LIN {X 0,Y 249.082,Z 599.459,A -85,B 0,C 180,E1 -18921.519,E2 -18921.519} C_VEL
LIN {X 0,Y 249.126,Z 599.438,A -85,B 0,C 180,E1 -18925.483,E2 -18925.483} C_VEL
LIN {X 0,Y 249.079,Z 599.446,A -85,B 0,C 180,E1 -18928.994,E2 -18928.994} C_VEL
LIN {X 0,Y 249.033,Z 599.465,A -85,B 0,C 180,E1 -18932.426,E2 -18932.426} C_VEL
LIN {X 0,Y 249.071,Z 599.46,A -85,B 0,C 180,E1 -18936.339,E2 -18936.339} C_VEL
LIN {X 0,Y 249.033,Z 599.471,A -85,B 0,C 180,E1 -18940.94,E2 -18940.94} C_VEL
LIN {X 0,Y 249.934,Z 602.079,A -85,B 0,C 180,E1 -18941.228,E2 -18941.228} C_VEL
LIN {X 0,Y 251.998,Z 604.708,A -85,B 0,C 180,E1 -18941.748,E2 -18941.748} C_VEL
LIN {X 0,Y 262.179,Z 620.888,A -85,B 0,C 180,E1 -18944.251,E2 -18944.251} C_VEL
LIN {X 0,Y 269.73,Z 634.216,A -85,B 0,C 180,E1 -18945.97,E2 -18945.97} C_VEL
LIN {X 0,Y 273.492,Z 641.681,A -85,B 0,C 180,E1 -18946.804,E2 -18946.804} C_VEL
LIN {X 0,Y 271.471,Z 691.803,A -85,B 0,C 180,E1 -18948.109,E2 -18948.109} C_VEL
LIN {X 0,Y 270.735,Z 705.187,A -85,B 0,C 180,E1 -18948.696,E2 -18948.696} C_VEL
LIN {X 0,Y 269.486,Z 718.044,A -85,B 0,C 180,E1 -18949.556,E2 -18949.556} C_VEL
LIN {X 0,Y 267.657,Z 730.406,A -85,B 0,C 180,E1 -18950.695,E2 -18950.695} C_VEL
LIN {X 0,Y 265.617,Z 741.459,A -85,B 0,C 180,E1 -18952.037,E2 -18952.037} C_VEL
LIN {X 0,Y 263.18,Z 752.351,A -85,B 0,C 180,E1 -18953.717,E2 -18953.717} C_VEL
LIN {X 0,Y 260.708,Z 761.621,A -85,B 0,C 180,E1 -18955.522,E2 -18955.522} C_VEL
LIN {X 0,Y 258.17,Z 770.535,A -85,B 0,C 180,E1 -18957.713,E2 -18957.713} C_VEL
LIN {X 0,Y 255.828,Z 777.697,A -85,B 0,C 180,E1 -18959.911,E2 -18959.911} C_VEL
LIN {X 0,Y 253.498,Z 784.302,A -85,B 0,C 180,E1 -18962.52,E2 -18962.52} C_VEL
LIN {X 0,Y 251.573,Z 789.492,A -85,B 0,C 180,E1 -18965.226,E2 -18965.226} C_VEL
LIN {X 0,Y 250.056,Z 793.37,A -85,B 0,C 180,E1 -18968.047,E2 -18968.047} C_VEL
LIN {X 0,Y 249.088,Z 795.421,A -85,B 0,C 180,E1 -18970.21,E2 -18970.21} C_VEL
LIN {X 0,Y 248.544,Z 796.494,A -85,B 0,C 180,E1 -18971.878,E2 -18971.878} C_VEL
LIN {X 0,Y 247.872,Z 797.374,A -85,B 0,C 180,E1 -18975.216,E2 -18975.216} C_VEL
LIN {X 0,Y 247.669,Z 797.218,A -85,B 0,C 180,E1 -18976.879,E2 -18976.879} C_VEL
LIN {X 0,Y 247.624,Z 795.63,A -85,B 0,C 180,E1 -18980.196,E2 -18980.196} C_VEL
LIN {X 0,Y 247.906,Z 793.165,A -85,B 0,C 180,E1 -18982.855,E2 -18982.855} C_VEL
LIN {X 0,Y 248.296,Z 790.13,A -85,B 0,C 180,E1 -18985.129,E2 -18985.129} C_VEL
LIN {X 0,Y 248.985,Z 785.826,A -85,B 0,C 180,E1 -18987.573,E2 -18987.573} C_VEL
LIN {X 0,Y 249.851,Z 780.356,A -85,B 0,C 180,E1 -18990,E2 -18990} C_VEL
LIN {X 0,Y 251.008,Z 773.505,A -85,B 0,C 180,E1 -18992.407,E2 -18992.407} C_VEL
LIN {X 0,Y 252.54,Z 764.911,A -85,B 0,C 180,E1 -18994.789,E2 -18994.789} C_VEL
LIN {X 0,Y 254.059,Z 756.117,A -85,B 0,C 180,E1 -18996.752,E2 -18996.752} C_VEL
LIN {X 0,Y 255.471,Z 746.489,A -85,B 0,C 180,E1 -18998.503,E2 -18998.503} C_VEL
LIN {X 0,Y 257.112,Z 734.896,A -85,B 0,C 180,E1 -19000.154,E2 -19000.154} C_VEL
LIN {X 0,Y 258.501,Z 722.796,A -85,B 0,C 180,E1 -19001.49,E2 -19001.49} C_VEL
LIN {X 0,Y 259.536,Z 710.236,A -85,B 0,C 180,E1 -19002.511,E2 -19002.511} C_VEL
LIN {X 0,Y 260.222,Z 696.894,A -85,B 0,C 180,E1 -19003.262,E2 -19003.262} C_VEL
LIN {X 0,Y 260.83,Z 676.4,A -85,B 0,C 180,E1 -19003.888,E2 -19003.888} C_VEL
LIN {X 0,Y 262.109,Z 629.666,A -85,B 0,C 180,E1 -19005.142,E2 -19005.142} C_VEL
LIN {X 0,Y 253.908,Z 610.003,A -85,B 0,C 180,E1 -19006.539,E2 -19006.539} C_VEL
LIN {X 0,Y 252.057,Z 606.531,A -85,B 0,C 180,E1 -19006.849,E2 -19006.849} C_VEL
LIN {X 0,Y 261.743,Z 629.406,A -85,B 0,C 180,E1 -19008.542,E2 -19008.542} C_VEL
LIN {X 0,Y 262.782,Z 631.947,A -85,B 0,C 180,E1 -19008.719,E2 -19008.719} C_VEL
LIN {X 0,Y 260.482,Z 693.854,A -85,B 0,C 180,E1 -19010.636,E2 -19010.636} C_VEL
LIN {X 0,Y 259.825,Z 707.287,A -85,B 0,C 180,E1 -19011.365,E2 -19011.365} C_VEL
LIN {X 0,Y 258.74,Z 719.997,A -85,B 0,C 180,E1 -19012.35,E2 -19012.35} C_VEL
LIN {X 0,Y 257.533,Z 731.237,A -85,B 0,C 180,E1 -19013.522,E2 -19013.522} C_VEL
LIN {X 0,Y 255.956,Z 743.817,A -85,B 0,C 180,E1 -19015.219,E2 -19015.219} C_VEL
LIN {X 0,Y 254.453,Z 753.674,A -85,B 0,C 180,E1 -19016.889,E2 -19016.889} C_VEL
LIN {X 0,Y 252.923,Z 763.074,A -85,B 0,C 180,E1 -19018.868,E2 -19018.868} C_VEL
LIN {X 0,Y 251.449,Z 771.778,A -85,B 0,C 180,E1 -19021.134,E2 -19021.134} C_VEL
LIN {X 0,Y 250.227,Z 778.82,A -85,B 0,C 180,E1 -19023.406,E2 -19023.406} C_VEL
LIN {X 0,Y 249.306,Z 784.585,A -85,B 0,C 180,E1 -19025.718,E2 -19025.718} C_VEL
LIN {X 0,Y 248.469,Z 789.922,A -85,B 0,C 180,E1 -19028.481,E2 -19028.481} C_VEL
LIN {X 0,Y 247.942,Z 793.177,A -85,B 0,C 180,E1 -19030.687,E2 -19030.687} C_VEL
LIN {X 0,Y 247.595,Z 795.616,A -85,B 0,C 180,E1 -19032.939,E2 -19032.939} C_VEL
LIN {X 0,Y 247.507,Z 797.247,A -85,B 0,C 180,E1 -19035.224,E2 -19035.224} C_VEL
LIN {X 0,Y 247.614,Z 798.097,A -85,B 0,C 180,E1 -19037.556,E2 -19037.556} C_VEL
LIN {X 0,Y 247.975,Z 798.121,A -85,B 0,C 180,E1 -19039.925,E2 -19039.925} C_VEL
LIN {X 0,Y 248.631,Z 797.271,A -85,B 0,C 180,E1 -19042.321,E2 -19042.321} C_VEL
LIN {X 0,Y 249.53,Z 795.476,A -85,B 0,C 180,E1 -19044.762,E2 -19044.762} C_VEL
LIN {X 0,Y 251.057,Z 791.727,A -85,B 0,C 180,E1 -19047.867,E2 -19047.867} C_VEL
LIN {X 0,Y 252.676,Z 787.333,A -85,B 0,C 180,E1 -19050.416,E2 -19050.416} C_VEL
LIN {X 0,Y 254.848,Z 781.199,A -85,B 0,C 180,E1 -19053.079,E2 -19053.079} C_VEL
LIN {X 0,Y 257.014,Z 774.612,A -85,B 0,C 180,E1 -19055.293,E2 -19055.293} C_VEL
LIN {X 0,Y 259.391,Z 766.758,A -85,B 0,C 180,E1 -19057.406,E2 -19057.406} C_VEL
LIN {X 0,Y 261.928,Z 757.594,A -85,B 0,C 180,E1 -19059.38,E2 -19059.38} C_VEL
LIN {X 0,Y 264.28,Z 747.756,A -85,B 0,C 180,E1 -19061.087,E2 -19061.087} C_VEL
LIN {X 0,Y 264.764,Z 743.074,A -85,B 0,C 180,E1 -19061.862,E2 -19061.862} C_VEL
LIN {X 0,Y 263.45,Z 732.357,A -85,B 0,C 180,E1 -19063.76,E2 -19063.76} C_VEL
LIN {X 0,Y 262.988,Z 725.778,A -85,B 0,C 180,E1 -19064.699,E2 -19064.699} C_VEL
LIN {X 0,Y 263.253,Z 722.241,A -85,B 0,C 180,E1 -19065.063,E2 -19065.063} C_VEL
LIN {X 0,Y 264.76,Z 709.401,A -85,B 0,C 180,E1 -19066.034,E2 -19066.034} C_VEL
LIN {X 0,Y 265.703,Z 696.323,A -85,B 0,C 180,E1 -19066.707,E2 -19066.707} C_VEL
LIN {X 0,Y 268.808,Z 643.586,A -85,B 0,C 180,E1 -19068.39,E2 -19068.39} C_VEL
LIN {X 0,Y 262.795,Z 631.883,A -85,B 0,C 180,E1 -19070.124,E2 -19070.124} C_VEL
LIN {X 0,Y 255.885,Z 620.412,A -85,B 0,C 180,E1 -19072.262,E2 -19072.262} C_VEL
LIN {X 0,Y 251.655,Z 613.959,A -85,B 0,C 180,E1 -19073.687,E2 -19073.687} C_VEL
LIN {X 0,Y 248.959,Z 610.142,A -85,B 0,C 180,E1 -19074.634,E2 -19074.634} C_VEL
LIN {X 0,Y 246.533,Z 607.111,A -85,B 0,C 180,E1 -19075.512,E2 -19075.512} C_VEL
LIN {X 0,Y 245.545,Z 605.398,A -85,B 0,C 180,E1 -19075.914,E2 -19075.914} C_VEL
LIN {X 0,Y 243.492,Z 603.287,A -85,B 0,C 180,E1 -19076.691,E2 -19076.691} C_VEL
LIN {X 0,Y 242.539,Z 600.953,A -85,B 0,C 180,E1 -19077.145,E2 -19077.145} C_VEL
LIN {X 0,Y 242.441,Z 600.281,A -85,B 0,C 180,E1 -19077.3,E2 -19077.3} C_VEL
LIN {X 0,Y 242.692,Z 600.249,A -85,B 0,C 180,E1 -19080,E2 -19080} C_VEL
LIN {X 0,Y 242.631,Z 600.261,A -85,B 0,C 180,E1 -19081.66,E2 -19081.66} C_VEL
LIN {X 0,Y 242.427,Z 600.277,A -85,B 0,C 180,E1 -19086.659,E2 -19086.659} C_VEL
LIN {X 0,Y 242.309,Z 600.288,A -85,B 0,C 180,E1 -19090.022,E2 -19090.022} C_VEL
LIN {X 0,Y 242.151,Z 600.315,A -85,B 0,C 180,E1 -19095.142,E2 -19095.142} C_VEL
LIN {X 0,Y 242.066,Z 600.326,A -85,B 0,C 180,E1 -19098.625,E2 -19098.625} C_VEL
LIN {X 0,Y 242.008,Z 600.337,A -85,B 0,C 180,E1 -19102.18,E2 -19102.18} C_VEL
LIN {X 0,Y 242.063,Z 600.334,A -85,B 0,C 180,E1 -19105.839,E2 -19105.839} C_VEL
LIN {X 0,Y 242.026,Z 600.335,A -85,B 0,C 180,E1 -19109.581,E2 -19109.581} C_VEL
LIN {X 0,Y 241.988,Z 600.335,A -85,B 0,C 180,E1 -19113.492,E2 -19113.492} C_VEL
LIN {X 0,Y 242.01,Z 600.338,A -85,B 0,C 180,E1 -19117.578,E2 -19117.578} C_VEL
LIN {X 0,Y 242.016,Z 600.535,A -85,B 0,C 180,E1 -19118.962,E2 -19118.962} C_VEL
LIN {X 0,Y 243.784,Z 605.815,A -85,B 0,C 180,E1 -19122.647,E2 -19122.647} C_VEL
LIN {X 0,Y 245.968,Z 612.642,A -85,B 0,C 180,E1 -19126.707,E2 -19126.707} C_VEL
LIN {X 0,Y 247.835,Z 619.474,A -85,B 0,C 180,E1 -19130.189,E2 -19130.189} C_VEL
LIN {X 0,Y 250.568,Z 624.665,A -85,B 0,C 180,E1 -19131.241,E2 -19131.241} C_VEL
LIN {X 0,Y 252.18,Z 627.583,A -85,B 0,C 180,E1 -19131.822,E2 -19131.822} C_VEL
LIN {X 0,Y 255.009,Z 632.985,A -85,B 0,C 180,E1 -19132.801,E2 -19132.801} C_VEL
LIN {X 0,Y 259.392,Z 642.122,A -85,B 0,C 180,E1 -19134.256,E2 -19134.256} C_VEL
LIN {X 0,Y 262.407,Z 649.312,A -85,B 0,C 180,E1 -19135.233,E2 -19135.233} C_VEL
LIN {X 0,Y 264.894,Z 668.043,A -85,B 0,C 180,E1 -19136.557,E2 -19136.557} C_VEL
LIN {X 0,Y 266.173,Z 683.879,A -85,B 0,C 180,E1 -19137.483,E2 -19137.483} C_VEL
LIN {X 0,Y 266.569,Z 690.964,A -85,B 0,C 180,E1 -19137.858,E2 -19137.858} C_VEL
LIN {X 0,Y 263.985,Z 733.939,A -85,B 0,C 180,E1 -19139.233,E2 -19139.233} C_VEL
LIN {X 0,Y 262.386,Z 747.924,A -85,B 0,C 180,E1 -19139.965,E2 -19139.965} C_VEL
LIN {X 0,Y 260.203,Z 760.61,A -85,B 0,C 180,E1 -19140.911,E2 -19140.911} C_VEL
LIN {X 0,Y 257.602,Z 772.84,A -85,B 0,C 180,E1 -19142.147,E2 -19142.147} C_VEL
LIN {X 0,Y 254.816,Z 783.944,A -85,B 0,C 180,E1 -19143.594,E2 -19143.594} C_VEL
LIN {X 0,Y 252.114,Z 794.049,A -85,B 0,C 180,E1 -19145.283,E2 -19145.283} C_VEL
LIN {X 0,Y 249.332,Z 803.305,A -85,B 0,C 180,E1 -19147.197,E2 -19147.197} C_VEL
LIN {X 0,Y 246.566,Z 812.457,A -85,B 0,C 180,E1 -19149.564,E2 -19149.564} C_VEL
LIN {X 0,Y 244.524,Z 819.897,A -85,B 0,C 180,E1 -19152.003,E2 -19152.003} C_VEL
LIN {X 0,Y 242.872,Z 824.973,A -85,B 0,C 180,E1 -19154.044,E2 -19154.044} C_VEL
LIN {X 0,Y 241.494,Z 829.974,A -85,B 0,C 180,E1 -19156.537,E2 -19156.537} C_VEL
LIN {X 0,Y 240.654,Z 833.88,A -85,B 0,C 180,E1 -19159.058,E2 -19159.058} C_VEL
LIN {X 0,Y 240.244,Z 836.788,A -85,B 0,C 180,E1 -19161.589,E2 -19161.589} C_VEL
LIN {X 0,Y 240.238,Z 838.715,A -85,B 0,C 180,E1 -19164.07,E2 -19164.07} C_VEL
LIN {X 0,Y 240.322,Z 839.767,A -85,B 0,C 180,E1 -19166.647,E2 -19166.647} C_VEL
LIN {X 0,Y 240.609,Z 839.94,A -85,B 0,C 180,E1 -19168.326,E2 -19168.326} C_VEL
LIN {X 0,Y 240.759,Z 839.692,A -85,B 0,C 180,E1 -19170,E2 -19170} C_VEL
LIN {X 0,Y 240.697,Z 838.969,A -85,B 0,C 180,E1 -19171.673,E2 -19171.673} C_VEL
LIN {X 0,Y 240.236,Z 837.756,A -85,B 0,C 180,E1 -19175.925,E2 -19175.925} C_VEL
LIN {X 0,Y 240.215,Z 836.024,A -85,B 0,C 180,E1 -19178.412,E2 -19178.412} C_VEL
LIN {X 0,Y 240.654,Z 833.336,A -85,B 0,C 180,E1 -19180.942,E2 -19180.942} C_VEL
LIN {X 0,Y 241.507,Z 829.65,A -85,B 0,C 180,E1 -19183.462,E2 -19183.462} C_VEL
LIN {X 0,Y 242.879,Z 824.868,A -85,B 0,C 180,E1 -19185.955,E2 -19185.955} C_VEL
LIN {X 0,Y 244.715,Z 818.848,A -85,B 0,C 180,E1 -19188.415,E2 -19188.415} C_VEL
LIN {X 0,Y 246.953,Z 811.391,A -85,B 0,C 180,E1 -19190.838,E2 -19190.838} C_VEL
LIN {X 0,Y 249.355,Z 803.827,A -85,B 0,C 180,E1 -19192.801,E2 -19192.801} C_VEL
LIN {X 0,Y 252.099,Z 794.685,A -85,B 0,C 180,E1 -19194.718,E2 -19194.718} C_VEL
LIN {X 0,Y 254.841,Z 784.535,A -85,B 0,C 180,E1 -19196.403,E2 -19196.403} C_VEL
LIN {X 0,Y 257.534,Z 773.315,A -85,B 0,C 180,E1 -19197.861,E2 -19197.861} C_VEL
LIN {X 0,Y 259.956,Z 761.689,A -85,B 0,C 180,E1 -19199.008,E2 -19199.008} C_VEL
LIN {X 0,Y 262.029,Z 748.941,A -85,B 0,C 180,E1 -19199.914,E2 -19199.914} C_VEL
LIN {X 0,Y 263.419,Z 735.313,A -85,B 0,C 180,E1 -19200.58,E2 -19200.58} C_VEL
LIN {X 0,Y 265.504,Z 686.502,A -85,B 0,C 180,E1 -19201.929,E2 -19201.929} C_VEL
LIN {X 0,Y 263.32,Z 661.252,A -85,B 0,C 180,E1 -19203.127,E2 -19203.127} C_VEL
LIN {X 0,Y 261.161,Z 643.82,A -85,B 0,C 180,E1 -19204.091,E2 -19204.091} C_VEL
LIN {X 0,Y 253.926,Z 625.793,A -85,B 0,C 180,E1 -19206.052,E2 -19206.052} C_VEL
LIN {X 0,Y 248.112,Z 612.261,A -85,B 0,C 180,E1 -19207.772,E2 -19207.772} C_VEL
LIN {X 0,Y 246.247,Z 608.323,A -85,B 0,C 180,E1 -19208.539,E2 -19208.539} C_VEL
LIN {X 0,Y 244.412,Z 604.945,A -85,B 0,C 180,E1 -19209.263,E2 -19209.263} C_VEL
LIN {X 0,Y 242.397,Z 601.9,A -85,B 0,C 180,E1 -19210.018,E2 -19210.018} C_VEL
LIN {X 0,Y 242.012,Z 600.339,A -85,B 0,C 180,E1 -19210.319,E2 -19210.319} C_VEL
LIN {X 0,Y 241.973,Z 600.343,A -85,B 0,C 180,E1 -19214.191,E2 -19214.191} C_VEL
LIN {X 0,Y 241.982,Z 600.344,A -85,B 0,C 180,E1 -19218.087,E2 -19218.087} C_VEL
LIN {X 0,Y 242.01,Z 600.339,A -85,B 0,C 180,E1 -19222.422,E2 -19222.422} C_VEL
LIN {X 0,Y 241.988,Z 600.327,A -85,B 0,C 180,E1 -19226.508,E2 -19226.508} C_VEL
LIN {X 0,Y 242.01,Z 600.318,A -85,B 0,C 180,E1 -19230.596,E2 -19230.596} C_VEL
LIN {X 0,Y 242.064,Z 600.334,A -85,B 0,C 180,E1 -19234.182,E2 -19234.182} C_VEL
LIN {X 0,Y 242.048,Z 600.313,A -85,B 0,C 180,E1 -19238.297,E2 -19238.297} C_VEL
LIN {X 0,Y 242.159,Z 600.297,A -85,B 0,C 180,E1 -19243.278,E2 -19243.278} C_VEL
LIN {X 0,Y 242.175,Z 600.316,A -85,B 0,C 180,E1 -19248.279,E2 -19248.279} C_VEL
LIN {X 0,Y 242.395,Z 600.264,A -85,B 0,C 180,E1 -19251.664,E2 -19251.664} C_VEL
LIN {X 0,Y 242.255,Z 600.308,A -85,B 0,C 180,E1 -19255.007,E2 -19255.007} C_VEL
LIN {X 0,Y 242.631,Z 600.233,A -85,B 0,C 180,E1 -19258.34,E2 -19258.34} C_VEL
LIN {X 0,Y 242.633,Z 600.261,A -85,B 0,C 180,E1 -19261.66,E2 -19261.66} C_VEL
LIN {X 0,Y 242.423,Z 600.264,A -85,B 0,C 180,E1 -19266.704,E2 -19266.704} C_VEL
LIN {X 0,Y 242.309,Z 600.3,A -85,B 0,C 180,E1 -19270.022,E2 -19270.022} C_VEL
LIN {X 0,Y 242.161,Z 600.318,A -85,B 0,C 180,E1 -19275.141,E2 -19275.141} C_VEL
LIN {X 0,Y 242.067,Z 600.311,A -85,B 0,C 180,E1 -19278.625,E2 -19278.625} C_VEL
LIN {X 0,Y 242.008,Z 600.34,A -85,B 0,C 180,E1 -19282.18,E2 -19282.18} C_VEL
LIN {X 0,Y 242.063,Z 600.32,A -85,B 0,C 180,E1 -19285.839,E2 -19285.839} C_VEL
LIN {X 0,Y 242.027,Z 600.321,A -85,B 0,C 180,E1 -19289.581,E2 -19289.581} C_VEL
LIN {X 0,Y 241.988,Z 600.333,A -85,B 0,C 180,E1 -19293.492,E2 -19293.492} C_VEL
LIN {X 0,Y 242.007,Z 600.337,A -85,B 0,C 180,E1 -19297.579,E2 -19297.579} C_VEL
LIN {X 0,Y 241.976,Z 600.444,A -85,B 0,C 180,E1 -19299.435,E2 -19299.435} C_VEL
LIN {X 0,Y 242.883,Z 603.039,A -85,B 0,C 180,E1 -19299.745,E2 -19299.745} C_VEL
LIN {X 0,Y 245.092,Z 605.693,A -85,B 0,C 180,E1 -19300.34,E2 -19300.34} C_VEL
LIN {X 0,Y 247.31,Z 609.082,A -85,B 0,C 180,E1 -19300.949,E2 -19300.949} C_VEL
LIN {X 0,Y 255.723,Z 622.291,A -85,B 0,C 180,E1 -19303.122,E2 -19303.122} C_VEL
LIN {X 0,Y 263.667,Z 636.132,A -85,B 0,C 180,E1 -19305.032,E2 -19305.032} C_VEL
LIN {X 0,Y 267.692,Z 644.022,A -85,B 0,C 180,E1 -19305.965,E2 -19305.965} C_VEL
LIN {X 0,Y 265.667,Z 692.159,A -85,B 0,C 180,E1 -19307.24,E2 -19307.24} C_VEL
LIN {X 0,Y 264.94,Z 704.98,A -85,B 0,C 180,E1 -19307.797,E2 -19307.797} C_VEL
LIN {X 0,Y 263.591,Z 718.518,A -85,B 0,C 180,E1 -19308.709,E2 -19308.709} C_VEL
LIN {X 0,Y 261.691,Z 730.922,A -85,B 0,C 180,E1 -19309.87,E2 -19309.87} C_VEL
LIN {X 0,Y 259.56,Z 741.989,A -85,B 0,C 180,E1 -19311.235,E2 -19311.235} C_VEL
LIN {X 0,Y 257.215,Z 752.039,A -85,B 0,C 180,E1 -19312.796,E2 -19312.796} C_VEL
LIN {X 0,Y 254.678,Z 761.285,A -85,B 0,C 180,E1 -19314.585,E2 -19314.585} C_VEL
LIN {X 0,Y 252,Z 770.255,A -85,B 0,C 180,E1 -19316.79,E2 -19316.79} C_VEL
LIN {X 0,Y 249.52,Z 777.661,A -85,B 0,C 180,E1 -19319.068,E2 -19319.068} C_VEL
LIN {X 0,Y 247.508,Z 783.074,A -85,B 0,C 180,E1 -19321.138,E2 -19321.138} C_VEL
LIN {X 0,Y 245.542,Z 788.295,A -85,B 0,C 180,E1 -19323.664,E2 -19323.664} C_VEL
LIN {X 0,Y 243.907,Z 792.268,A -85,B 0,C 180,E1 -19326.21,E2 -19326.21} C_VEL
LIN {X 0,Y 243.024,Z 794.273,A -85,B 0,C 180,E1 -19327.918,E2 -19327.918} C_VEL
LIN {X 0,Y 242.241,Z 795.843,A -85,B 0,C 180,E1 -19329.626,E2 -19329.626} C_VEL
LIN {X 0,Y 241.64,Z 796.994,A -85,B 0,C 180,E1 -19331.342,E2 -19331.342} C_VEL
LIN {X 0,Y 240.976,Z 797.93,A -85,B 0,C 180,E1 -19334.246,E2 -19334.246} C_VEL
LIN {X 0,Y 240.626,Z 797.865,A -85,B 0,C 180,E1 -19336.488,E2 -19336.488} C_VEL
LIN {X 0,Y 240.506,Z 797.337,A -85,B 0,C 180,E1 -19338.197,E2 -19338.197} C_VEL
LIN {X 0,Y 240.533,Z 796.388,A -85,B 0,C 180,E1 -19339.904,E2 -19339.904} C_VEL
LIN {X 0,Y 240.825,Z 793.784,A -85,B 0,C 180,E1 -19342.852,E2 -19342.852} C_VEL
LIN {X 0,Y 241.404,Z 789.793,A -85,B 0,C 180,E1 -19345.826,E2 -19345.826} C_VEL
LIN {X 0,Y 242.087,Z 785.213,A -85,B 0,C 180,E1 -19348.336,E2 -19348.336} C_VEL
LIN {X 0,Y 243.317,Z 778.3,A -85,B 0,C 180,E1 -19351.241,E2 -19351.241} C_VEL
LIN {X 0,Y 244.659,Z 770.804,A -85,B 0,C 180,E1 -19353.706,E2 -19353.706} C_VEL
LIN {X 0,Y 246.398,Z 761.368,A -85,B 0,C 180,E1 -19356.14,E2 -19356.14} C_VEL
LIN {X 0,Y 248.009,Z 751.67,A -85,B 0,C 180,E1 -19358.145,E2 -19358.145} C_VEL
LIN {X 0,Y 249.439,Z 742.114,A -85,B 0,C 180,E1 -19359.732,E2 -19359.732} C_VEL
LIN {X 0,Y 251.084,Z 730.087,A -85,B 0,C 180,E1 -19361.299,E2 -19361.299} C_VEL
LIN {X 0,Y 252.426,Z 717.413,A -85,B 0,C 180,E1 -19362.55,E2 -19362.55} C_VEL
LIN {X 0,Y 253.326,Z 703.996,A -85,B 0,C 180,E1 -19363.493,E2 -19363.493} C_VEL
LIN {X 0,Y 253.825,Z 692.175,A -85,B 0,C 180,E1 -19364.034,E2 -19364.034} C_VEL
LIN {X 0,Y 255.543,Z 631.329,A -85,B 0,C 180,E1 -19365.723,E2 -19365.723} C_VEL
LIN {X 0,Y 249.572,Z 617.012,A -85,B 0,C 180,E1 -19366.774,E2 -19366.774} C_VEL
LIN {X 0,Y 248.967,Z 616.257,A -85,B 0,C 180,E1 -19366.891,E2 -19366.891} C_VEL
LIN {X 0,Y 256.056,Z 633.482,A -85,B 0,C 180,E1 -19368.175,E2 -19368.175} C_VEL
LIN {X 0,Y 253.758,Z 694.75,A -85,B 0,C 180,E1 -19370.135,E2 -19370.135} C_VEL
LIN {X 0,Y 253.112,Z 707.921,A -85,B 0,C 180,E1 -19370.874,E2 -19370.874} C_VEL
LIN {X 0,Y 251.945,Z 720.869,A -85,B 0,C 180,E1 -19371.906,E2 -19371.906} C_VEL
LIN {X 0,Y 250.712,Z 732.028,A -85,B 0,C 180,E1 -19373.106,E2 -19373.106} C_VEL
LIN {X 0,Y 249.1,Z 744.362,A -85,B 0,C 180,E1 -19374.814,E2 -19374.814} C_VEL
LIN {X 0,Y 247.506,Z 754.515,A -85,B 0,C 180,E1 -19376.582,E2 -19376.582} C_VEL
LIN {X 0,Y 245.871,Z 764.364,A -85,B 0,C 180,E1 -19378.735,E2 -19378.735} C_VEL
LIN {X 0,Y 244.314,Z 773.36,A -85,B 0,C 180,E1 -19381.183,E2 -19381.183} C_VEL
LIN {X 0,Y 242.925,Z 781.023,A -85,B 0,C 180,E1 -19383.842,E2 -19383.842} C_VEL
LIN {X 0,Y 241.944,Z 787.212,A -85,B 0,C 180,E1 -19386.589,E2 -19386.589} C_VEL
LIN {X 0,Y 241.273,Z 791.378,A -85,B 0,C 180,E1 -19388.978,E2 -19388.978} C_VEL
LIN {X 0,Y 240.875,Z 793.734,A -85,B 0,C 180,E1 -19390.659,E2 -19390.659} C_VEL
LIN {X 0,Y 240.526,Z 796.285,A -85,B 0,C 180,E1 -19393.073,E2 -19393.073} C_VEL
LIN {X 0,Y 240.449,Z 797.924,A -85,B 0,C 180,E1 -19395.453,E2 -19395.453} C_VEL
LIN {X 0,Y 240.573,Z 798.742,A -85,B 0,C 180,E1 -19397.785,E2 -19397.785} C_VEL
LIN {X 0,Y 240.934,Z 798.803,A -85,B 0,C 180,E1 -19400.078,E2 -19400.078} C_VEL
LIN {X 0,Y 241.56,Z 798.11,A -85,B 0,C 180,E1 -19402.34,E2 -19402.34} C_VEL
LIN {X 0,Y 242.87,Z 795.706,A -85,B 0,C 180,E1 -19405.648,E2 -19405.648} C_VEL
LIN {X 0,Y 244.581,Z 791.753,A -85,B 0,C 180,E1 -19408.853,E2 -19408.853} C_VEL
LIN {X 0,Y 246.464,Z 786.944,A -85,B 0,C 180,E1 -19411.546,E2 -19411.546} C_VEL
LIN {X 0,Y 248.453,Z 781.572,A -85,B 0,C 180,E1 -19413.853,E2 -19413.853} C_VEL
LIN {X 0,Y 251.19,Z 773.662,A -85,B 0,C 180,E1 -19416.503,E2 -19416.503} C_VEL
LIN {X 0,Y 253.53,Z 766.278,A -85,B 0,C 180,E1 -19418.464,E2 -19418.464} C_VEL
LIN {X 0,Y 256.317,Z 756.621,A -85,B 0,C 180,E1 -19420.513,E2 -19420.513} C_VEL
LIN {X 0,Y 258.867,Z 746.072,A -85,B 0,C 180,E1 -19422.297,E2 -19422.297} C_VEL
LIN {X 0,Y 261.219,Z 734.806,A -85,B 0,C 180,E1 -19423.791,E2 -19423.791} C_VEL
LIN {X 0,Y 263.253,Z 722.241,A -85,B 0,C 180,E1 -19425.063,E2 -19425.063} C_VEL
LIN {X 0,Y 263.437,Z 716.858,A -85,B 0,C 180,E1 -19425.604,E2 -19425.604} C_VEL
LIN {X 0,Y 262.062,Z 708.191,A -85,B 0,C 180,E1 -19426.634,E2 -19426.634} C_VEL
LIN {X 0,Y 260.566,Z 699.306,A -85,B 0,C 180,E1 -19427.517,E2 -19427.517} C_VEL
LIN {X 0,Y 260.507,Z 693.606,A -85,B 0,C 180,E1 -19427.815,E2 -19427.815} C_VEL
LIN {X 0,Y 263.356,Z 646.129,A -85,B 0,C 180,E1 -19429.355,E2 -19429.355} C_VEL
LIN {X 0,Y 258.193,Z 635.958,A -85,B 0,C 180,E1 -19430.952,E2 -19430.952} C_VEL
LIN {X 0,Y 251.771,Z 625.024,A -85,B 0,C 180,E1 -19433.065,E2 -19433.065} C_VEL
LIN {X 0,Y 247.739,Z 618.869,A -85,B 0,C 180,E1 -19434.495,E2 -19434.495} C_VEL
LIN {X 0,Y 245.452,Z 615.654,A -85,B 0,C 180,E1 -19435.336,E2 -19435.336} C_VEL
LIN {X 0,Y 243.075,Z 612.405,A -85,B 0,C 180,E1 -19436.27,E2 -19436.27} C_VEL
LIN {X 0,Y 242.084,Z 611.047,A -85,B 0,C 180,E1 -19436.671,E2 -19436.671} C_VEL
LIN {X 0,Y 239.913,Z 608.252,A -85,B 0,C 180,E1 -19437.566,E2 -19437.566} C_VEL
LIN {X 0,Y 238.879,Z 606.324,A -85,B 0,C 180,E1 -19438.054,E2 -19438.054} C_VEL
LIN {X 0,Y 236.616,Z 604.003,A -85,B 0,C 180,E1 -19439.043,E2 -19439.043} C_VEL
LIN {X 0,Y 235.682,Z 601.577,A -85,B 0,C 180,E1 -19439.573,E2 -19439.573} C_VEL
LIN {X 0,Y 235.637,Z 601.13,A -85,B 0,C 180,E1 -19439.68,E2 -19439.68} C_VEL
LIN {X 0,Y 235.591,Z 601.138,A -85,B 0,C 180,E1 -19441.709,E2 -19441.709} C_VEL
LIN {X 0,Y 235.398,Z 601.152,A -85,B 0,C 180,E1 -19446.859,E2 -19446.859} C_VEL
LIN {X 0,Y 235.233,Z 601.169,A -85,B 0,C 180,E1 -19450.327,E2 -19450.327} C_VEL
LIN {X 0,Y 235.102,Z 601.192,A -85,B 0,C 180,E1 -19455.607,E2 -19455.607} C_VEL
LIN {X 0,Y 235.002,Z 601.205,A -85,B 0,C 180,E1 -19459.206,E2 -19459.206} C_VEL
LIN {X 0,Y 234.957,Z 601.212,A -85,B 0,C 180,E1 -19462.883,E2 -19462.883} C_VEL
LIN {X 0,Y 234.966,Z 601.21,A -85,B 0,C 180,E1 -19466.658,E2 -19466.658} C_VEL
LIN {X 0,Y 234.928,Z 601.214,A -85,B 0,C 180,E1 -19470.568,E2 -19470.568} C_VEL
LIN {X 0,Y 234.957,Z 601.214,A -85,B 0,C 180,E1 -19474.634,E2 -19474.634} C_VEL
LIN {X 0,Y 234.966,Z 601.275,A -85,B 0,C 180,E1 -19476.365,E2 -19476.365} C_VEL
LIN {X 0,Y 236.113,Z 604.842,A -85,B 0,C 180,E1 -19479.296,E2 -19479.296} C_VEL
LIN {X 0,Y 237.787,Z 609.78,A -85,B 0,C 180,E1 -19482.827,E2 -19482.827} C_VEL
LIN {X 0,Y 239.969,Z 616.822,A -85,B 0,C 180,E1 -19487.07,E2 -19487.07} C_VEL
LIN {X 0,Y 240.407,Z 618.341,A -85,B 0,C 180,E1 -19487.873,E2 -19487.873} C_VEL
LIN {X 0,Y 243.522,Z 623.893,A -85,B 0,C 180,E1 -19489.197,E2 -19489.197} C_VEL
LIN {X 0,Y 244.769,Z 626.089,A -85,B 0,C 180,E1 -19489.703,E2 -19489.703} C_VEL
LIN {X 0,Y 248.17,Z 632.193,A -85,B 0,C 180,E1 -19490.998,E2 -19490.998} C_VEL
LIN {X 0,Y 251.648,Z 639.199,A -85,B 0,C 180,E1 -19492.29,E2 -19492.29} C_VEL
LIN {X 0,Y 256.589,Z 650.047,A -85,B 0,C 180,E1 -19493.999,E2 -19493.999} C_VEL
LIN {X 0,Y 257.629,Z 653.231,A -85,B 0,C 180,E1 -19494.387,E2 -19494.387} C_VEL
LIN {X 0,Y 259.927,Z 672.484,A -85,B 0,C 180,E1 -19495.77,E2 -19495.77} C_VEL
LIN {X 0,Y 261.188,Z 690.853,A -85,B 0,C 180,E1 -19496.837,E2 -19496.837} C_VEL
LIN {X 0,Y 258.49,Z 733.294,A -85,B 0,C 180,E1 -19498.236,E2 -19498.236} C_VEL
LIN {X 0,Y 256.927,Z 746.254,A -85,B 0,C 180,E1 -19498.916,E2 -19498.916} C_VEL
LIN {X 0,Y 254.868,Z 758.156,A -85,B 0,C 180,E1 -19499.786,E2 -19499.786} C_VEL
LIN {X 0,Y 252.114,Z 770.759,A -85,B 0,C 180,E1 -19501.031,E2 -19501.031} C_VEL
LIN {X 0,Y 249.248,Z 782.101,A -85,B 0,C 180,E1 -19502.502,E2 -19502.502} C_VEL
LIN {X 0,Y 246.299,Z 792.467,A -85,B 0,C 180,E1 -19504.206,E2 -19504.206} C_VEL
LIN {X 0,Y 243.386,Z 801.881,A -85,B 0,C 180,E1 -19506.156,E2 -19506.156} C_VEL
LIN {X 0,Y 240.359,Z 811.115,A -85,B 0,C 180,E1 -19508.563,E2 -19508.563} C_VEL
LIN {X 0,Y 238.065,Z 818.642,A -85,B 0,C 180,E1 -19511.051,E2 -19511.051} C_VEL
LIN {X 0,Y 236.012,Z 824.776,A -85,B 0,C 180,E1 -19513.567,E2 -19513.567} C_VEL
LIN {X 0,Y 234.568,Z 829.685,A -85,B 0,C 180,E1 -19516.132,E2 -19516.132} C_VEL
LIN {X 0,Y 233.619,Z 833.506,A -85,B 0,C 180,E1 -19518.724,E2 -19518.724} C_VEL
LIN {X 0,Y 233.189,Z 836.324,A -85,B 0,C 180,E1 -19521.333,E2 -19521.333} C_VEL
LIN {X 0,Y 233.169,Z 838.282,A -85,B 0,C 180,E1 -19524.079,E2 -19524.079} C_VEL
LIN {X 0,Y 233.244,Z 839.153,A -85,B 0,C 180,E1 -19526.545,E2 -19526.545} C_VEL
LIN {X 0,Y 233.529,Z 839.292,A -85,B 0,C 180,E1 -19528.275,E2 -19528.275} C_VEL
LIN {X 0,Y 233.704,Z 838.998,A -85,B 0,C 180,E1 -19530,E2 -19530} C_VEL
LIN {X 0,Y 233.632,Z 838.215,A -85,B 0,C 180,E1 -19531.724,E2 -19531.724} C_VEL
LIN {X 0,Y 233.165,Z 837.31,A -85,B 0,C 180,E1 -19535.912,E2 -19535.912} C_VEL
LIN {X 0,Y 233.167,Z 835.527,A -85,B 0,C 180,E1 -19538.668,E2 -19538.668} C_VEL
LIN {X 0,Y 233.621,Z 832.889,A -85,B 0,C 180,E1 -19541.276,E2 -19541.276} C_VEL
LIN {X 0,Y 234.581,Z 829.262,A -85,B 0,C 180,E1 -19543.867,E2 -19543.867} C_VEL
LIN {X 0,Y 236.021,Z 824.541,A -85,B 0,C 180,E1 -19546.432,E2 -19546.432} C_VEL
LIN {X 0,Y 238.049,Z 818.124,A -85,B 0,C 180,E1 -19549.135,E2 -19549.135} C_VEL
LIN {X 0,Y 240.311,Z 811.212,A -85,B 0,C 180,E1 -19551.442,E2 -19551.442} C_VEL
LIN {X 0,Y 243.382,Z 802.102,A -85,B 0,C 180,E1 -19553.845,E2 -19553.845} C_VEL
LIN {X 0,Y 246.629,Z 791.591,A -85,B 0,C 180,E1 -19555.984,E2 -19555.984} C_VEL
LIN {X 0,Y 249.542,Z 780.925,A -85,B 0,C 180,E1 -19557.69,E2 -19557.69} C_VEL
LIN {X 0,Y 252.079,Z 770.564,A -85,B 0,C 180,E1 -19558.973,E2 -19558.973} C_VEL
LIN {X 0,Y 254.567,Z 758.151,A -85,B 0,C 180,E1 -19560.139,E2 -19560.139} C_VEL
LIN {X 0,Y 256.636,Z 745.097,A -85,B 0,C 180,E1 -19561.009,E2 -19561.009} C_VEL
LIN {X 0,Y 257.801,Z 732.249,A -85,B 0,C 180,E1 -19561.58,E2 -19561.58} C_VEL
LIN {X 0,Y 259.757,Z 687.067,A -85,B 0,C 180,E1 -19562.837,E2 -19562.837} C_VEL
LIN {X 0,Y 257.73,Z 662.922,A -85,B 0,C 180,E1 -19564.023,E2 -19564.023} C_VEL
LIN {X 0,Y 255.864,Z 646.747,A -85,B 0,C 180,E1 -19564.932,E2 -19564.932} C_VEL
LIN {X 0,Y 249.332,Z 630.114,A -85,B 0,C 180,E1 -19566.791,E2 -19566.791} C_VEL
LIN {X 0,Y 243.042,Z 615.654,A -85,B 0,C 180,E1 -19568.67,E2 -19568.67} C_VEL
LIN {X 0,Y 241.1,Z 612.498,A -85,B 0,C 180,E1 -19569.241,E2 -19569.241} C_VEL
LIN {X 0,Y 238.786,Z 608.604,A -85,B 0,C 180,E1 -19570.162,E2 -19570.162} C_VEL
LIN {X 0,Y 236.901,Z 605.31,A -85,B 0,C 180,E1 -19570.95,E2 -19570.95} C_VEL
LIN {X 0,Y 235.217,Z 602.467,A -85,B 0,C 180,E1 -19571.671,E2 -19571.671} C_VEL
LIN {X 0,Y 234.928,Z 601.211,A -85,B 0,C 180,E1 -19571.956,E2 -19571.956} C_VEL
LIN {X 0,Y 234.963,Z 601.206,A -85,B 0,C 180,E1 -19576.531,E2 -19576.531} C_VEL
LIN {X 0,Y 234.952,Z 601.205,A -85,B 0,C 180,E1 -19581.085,E2 -19581.085} C_VEL
LIN {X 0,Y 234.957,Z 601.197,A -85,B 0,C 180,E1 -19585.366,E2 -19585.366} C_VEL
LIN {X 0,Y 234.92,Z 601.212,A -85,B 0,C 180,E1 -19589.43,E2 -19589.43} C_VEL
LIN {X 0,Y 234.99,Z 601.213,A -85,B 0,C 180,E1 -19593.793,E2 -19593.793} C_VEL
LIN {X 0,Y 235.007,Z 601.197,A -85,B 0,C 180,E1 -19598.969,E2 -19598.969} C_VEL
LIN {X 0,Y 235.091,Z 601.179,A -85,B 0,C 180,E1 -19603.06,E2 -19603.06} C_VEL
LIN {X 0,Y 235.108,Z 601.199,A -85,B 0,C 180,E1 -19607.922,E2 -19607.922} C_VEL
LIN {X 0,Y 235.326,Z 601.143,A -85,B 0,C 180,E1 -19611.412,E2 -19611.412} C_VEL
LIN {X 0,Y 235.369,Z 601.154,A -85,B 0,C 180,E1 -19613.14,E2 -19613.14} C_VEL
LIN {X 0,Y 235.591,Z 601.11,A -85,B 0,C 180,E1 -19618.291,E2 -19618.291} C_VEL
LIN {X 0,Y 235.593,Z 601.138,A -85,B 0,C 180,E1 -19621.709,E2 -19621.709} C_VEL
LIN {X 0,Y 235.397,Z 601.14,A -85,B 0,C 180,E1 -19626.859,E2 -19626.859} C_VEL
LIN {X 0,Y 235.233,Z 601.176,A -85,B 0,C 180,E1 -19630.327,E2 -19630.327} C_VEL
LIN {X 0,Y 235.109,Z 601.199,A -85,B 0,C 180,E1 -19635.607,E2 -19635.607} C_VEL
LIN {X 0,Y 235.003,Z 601.19,A -85,B 0,C 180,E1 -19639.206,E2 -19639.206} C_VEL
LIN {X 0,Y 234.956,Z 601.212,A -85,B 0,C 180,E1 -19642.883,E2 -19642.883} C_VEL
LIN {X 0,Y 234.966,Z 601.214,A -85,B 0,C 180,E1 -19646.658,E2 -19646.658} C_VEL
LIN {X 0,Y 234.929,Z 601.207,A -85,B 0,C 180,E1 -19650.568,E2 -19650.568} C_VEL
LIN {X 0,Y 234.957,Z 601.205,A -85,B 0,C 180,E1 -19654.634,E2 -19654.634} C_VEL
LIN {X 0,Y 234.965,Z 601.214,A -85,B 0,C 180,E1 -19657.785,E2 -19657.785} C_VEL
LIN {X 0,Y 235.981,Z 604.088,A -85,B 0,C 180,E1 -19658.169,E2 -19658.169} C_VEL
LIN {X 0,Y 238.151,Z 606.675,A -85,B 0,C 180,E1 -19658.801,E2 -19658.801} C_VEL
LIN {X 0,Y 240.436,Z 610.111,A -85,B 0,C 180,E1 -19659.476,E2 -19659.476} C_VEL
LIN {X 0,Y 246.629,Z 619.388,A -85,B 0,C 180,E1 -19661.205,E2 -19661.205} C_VEL
LIN {X 0,Y 254.591,Z 632.586,A -85,B 0,C 180,E1 -19663.281,E2 -19663.281} C_VEL
LIN {X 0,Y 261.432,Z 645.326,A -85,B 0,C 180,E1 -19664.965,E2 -19664.965} C_VEL
LIN {X 0,Y 261.979,Z 646.386,A -85,B 0,C 180,E1 -19665.095,E2 -19665.095} C_VEL
LIN {X 0,Y 259.945,Z 692.558,A -85,B 0,C 180,E1 -19666.337,E2 -19666.337} C_VEL
LIN {X 0,Y 259.156,Z 705.616,A -85,B 0,C 180,E1 -19666.909,E2 -19666.909} C_VEL
LIN {X 0,Y 257.857,Z 718.165,A -85,B 0,C 180,E1 -19667.758,E2 -19667.758} C_VEL
LIN {X 0,Y 256.096,Z 729.641,A -85,B 0,C 180,E1 -19668.806,E2 -19668.806} C_VEL
LIN {X 0,Y 253.871,Z 741.112,A -85,B 0,C 180,E1 -19670.196,E2 -19670.196} C_VEL
LIN {X 0,Y 251.094,Z 752.642,A -85,B 0,C 180,E1 -19671.993,E2 -19671.993} C_VEL
LIN {X 0,Y 248.197,Z 762.746,A -85,B 0,C 180,E1 -19674.017,E2 -19674.017} C_VEL
LIN {X 0,Y 245.291,Z 771.876,A -85,B 0,C 180,E1 -19676.354,E2 -19676.354} C_VEL
LIN {X 0,Y 242.815,Z 778.85,A -85,B 0,C 180,E1 -19678.602,E2 -19678.602} C_VEL
LIN {X 0,Y 240.158,Z 785.586,A -85,B 0,C 180,E1 -19681.393,E2 -19681.393} C_VEL
LIN {X 0,Y 238.363,Z 789.967,A -85,B 0,C 180,E1 -19683.752,E2 -19683.752} C_VEL
LIN {X 0,Y 236.668,Z 793.756,A -85,B 0,C 180,E1 -19686.46,E2 -19686.46} C_VEL
LIN {X 0,Y 235.427,Z 796.265,A -85,B 0,C 180,E1 -19689.009,E2 -19689.009} C_VEL
LIN {X 0,Y 234.746,Z 797.465,A -85,B 0,C 180,E1 -19690.773,E2 -19690.773} C_VEL
LIN {X 0,Y 233.946,Z 798.539,A -85,B 0,C 180,E1 -19694.012,E2 -19694.012} C_VEL
LIN {X 0,Y 233.606,Z 798.498,A -85,B 0,C 180,E1 -19696.074,E2 -19696.074} C_VEL
LIN {X 0,Y 233.439,Z 798.047,A -85,B 0,C 180,E1 -19697.834,E2 -19697.834} C_VEL
LIN {X 0,Y 233.463,Z 797.144,A -85,B 0,C 180,E1 -19699.594,E2 -19699.594} C_VEL
LIN {X 0,Y 233.748,Z 794.412,A -85,B 0,C 180,E1 -19702.839,E2 -19702.839} C_VEL
LIN {X 0,Y 234.292,Z 790.747,A -85,B 0,C 180,E1 -19705.699,E2 -19705.699} C_VEL
LIN {X 0,Y 234.989,Z 786.275,A -85,B 0,C 180,E1 -19708.286,E2 -19708.286} C_VEL
LIN {X 0,Y 236.237,Z 779.473,A -85,B 0,C 180,E1 -19711.278,E2 -19711.278} C_VEL
LIN {X 0,Y 237.593,Z 772.122,A -85,B 0,C 180,E1 -19713.816,E2 -19713.816} C_VEL
LIN {X 0,Y 239.058,Z 764.592,A -85,B 0,C 180,E1 -19715.906,E2 -19715.906} C_VEL
LIN {X 0,Y 240.85,Z 754.395,A -85,B 0,C 180,E1 -19718.178,E2 -19718.178} C_VEL
LIN {X 0,Y 242.483,Z 744.072,A -85,B 0,C 180,E1 -19720.014,E2 -19720.014} C_VEL
LIN {X 0,Y 244.168,Z 732.452,A -85,B 0,C 180,E1 -19721.623,E2 -19721.623} C_VEL
LIN {X 0,Y 245.561,Z 720.354,A -85,B 0,C 180,E1 -19722.904,E2 -19722.904} C_VEL
LIN {X 0,Y 246.556,Z 707.563,A -85,B 0,C 180,E1 -19723.902,E2 -19723.902} C_VEL
LIN {X 0,Y 247.233,Z 693.77,A -85,B 0,C 180,E1 -19724.594,E2 -19724.594} C_VEL
LIN {X 0,Y 249.003,Z 633.01,A -85,B 0,C 180,E1 -19726.334,E2 -19726.334} C_VEL
LIN {X 0,Y 246.424,Z 626.878,A -85,B 0,C 180,E1 -19726.798,E2 -19726.798} C_VEL
LIN {X 0,Y 245.73,Z 625.944,A -85,B 0,C 180,E1 -19726.918,E2 -19726.918} C_VEL
LIN {X 0,Y 249.499,Z 635.748,A -85,B 0,C 180,E1 -19727.641,E2 -19727.641} C_VEL
LIN {X 0,Y 247.099,Z 695.259,A -85,B 0,C 180,E1 -19729.591,E2 -19729.591} C_VEL
LIN {X 0,Y 246.38,Z 708.777,A -85,B 0,C 180,E1 -19730.37,E2 -19730.37} C_VEL
LIN {X 0,Y 245.179,Z 721.714,A -85,B 0,C 180,E1 -19731.436,E2 -19731.436} C_VEL
LIN {X 0,Y 243.671,Z 734.639,A -85,B 0,C 180,E1 -19732.9,E2 -19732.9} C_VEL
LIN {X 0,Y 242.232,Z 745.132,A -85,B 0,C 180,E1 -19734.421,E2 -19734.421} C_VEL
LIN {X 0,Y 240.608,Z 755.152,A -85,B 0,C 180,E1 -19736.217,E2 -19736.217} C_VEL
LIN {X 0,Y 238.862,Z 765.517,A -85,B 0,C 180,E1 -19738.561,E2 -19738.561} C_VEL
LIN {X 0,Y 237.2,Z 774.522,A -85,B 0,C 180,E1 -19741.115,E2 -19741.115} C_VEL
LIN {X 0,Y 235.783,Z 782.314,A -85,B 0,C 180,E1 -19743.948,E2 -19743.948} C_VEL
LIN {X 0,Y 234.774,Z 788.373,A -85,B 0,C 180,E1 -19746.776,E2 -19746.776} C_VEL
LIN {X 0,Y 234.161,Z 792.165,A -85,B 0,C 180,E1 -19749.07,E2 -19749.07} C_VEL
LIN {X 0,Y 233.631,Z 795.194,A -85,B 0,C 180,E1 -19751.436,E2 -19751.436} C_VEL
LIN {X 0,Y 233.407,Z 797.414,A -85,B 0,C 180,E1 -19753.83,E2 -19753.83} C_VEL
LIN {X 0,Y 233.405,Z 798.864,A -85,B 0,C 180,E1 -19756.273,E2 -19756.273} C_VEL
LIN {X 0,Y 233.621,Z 799.511,A -85,B 0,C 180,E1 -19758.768,E2 -19758.768} C_VEL
LIN {X 0,Y 234.178,Z 799.28,A -85,B 0,C 180,E1 -19761.286,E2 -19761.286} C_VEL
LIN {X 0,Y 235.018,Z 798.164,A -85,B 0,C 180,E1 -19763.842,E2 -19763.842} C_VEL
LIN {X 0,Y 236.154,Z 796.088,A -85,B 0,C 180,E1 -19766.435,E2 -19766.435} C_VEL
LIN {X 0,Y 237.637,Z 792.946,A -85,B 0,C 180,E1 -19769.052,E2 -19769.052} C_VEL
LIN {X 0,Y 239.737,Z 787.987,A -85,B 0,C 180,E1 -19772.027,E2 -19772.027} C_VEL
LIN {X 0,Y 242.223,Z 781.722,A -85,B 0,C 180,E1 -19774.78,E2 -19774.78} C_VEL
LIN {X 0,Y 244.725,Z 774.965,A -85,B 0,C 180,E1 -19777.094,E2 -19777.094} C_VEL
LIN {X 0,Y 247.641,Z 766.215,A -85,B 0,C 180,E1 -19779.473,E2 -19779.473} C_VEL
LIN {X 0,Y 250.642,Z 756.066,A -85,B 0,C 180,E1 -19781.613,E2 -19781.613} C_VEL
LIN {X 0,Y 253.495,Z 744.804,A -85,B 0,C 180,E1 -19783.49,E2 -19783.49} C_VEL
LIN {X 0,Y 256.045,Z 732.567,A -85,B 0,C 180,E1 -19785.055,E2 -19785.055} C_VEL
LIN {X 0,Y 258.043,Z 720.69,A -85,B 0,C 180,E1 -19786.211,E2 -19786.211} C_VEL
LIN {X 0,Y 259.499,Z 707.672,A -85,B 0,C 180,E1 -19787.152,E2 -19787.152} C_VEL
LIN {X 0,Y 260.45,Z 694.458,A -85,B 0,C 180,E1 -19787.785,E2 -19787.785} C_VEL
LIN {X 0,Y 260.507,Z 693.606,A -85,B 0,C 180,E1 -19787.815,E2 -19787.815} C_VEL
LIN {X 0,Y 260.447,Z 687.841,A -85,B 0,C 180,E1 -19788.081,E2 -19788.081} C_VEL
LIN {X 0,Y 257.323,Z 669.419,A -85,B 0,C 180,E1 -19789.553,E2 -19789.553} C_VEL
LIN {X 0,Y 257.188,Z 663.661,A -85,B 0,C 180,E1 -19789.852,E2 -19789.852} C_VEL
LIN {X 0,Y 258.129,Z 648.77,A -85,B 0,C 180,E1 -19790.353,E2 -19790.353} C_VEL
LIN {X 0,Y 253.309,Z 639.272,A -85,B 0,C 180,E1 -19791.933,E2 -19791.933} C_VEL
LIN {X 0,Y 246.792,Z 628.161,A -85,B 0,C 180,E1 -19794.241,E2 -19794.241} C_VEL
LIN {X 0,Y 242.491,Z 621.648,A -85,B 0,C 180,E1 -19795.897,E2 -19795.897} C_VEL
LIN {X 0,Y 239.758,Z 617.828,A -85,B 0,C 180,E1 -19797.015,E2 -19797.015} C_VEL
LIN {X 0,Y 236.684,Z 613.667,A -85,B 0,C 180,E1 -19798.352,E2 -19798.352} C_VEL
LIN {X 0,Y 235.703,Z 612.127,A -85,B 0,C 180,E1 -19798.825,E2 -19798.825} C_VEL
LIN {X 0,Y 233.462,Z 609.359,A -85,B 0,C 180,E1 -19799.892,E2 -19799.892} C_VEL
LIN {X 0,Y 232.639,Z 607.569,A -85,B 0,C 180,E1 -19800.357,E2 -19800.357} C_VEL
LIN {X 0,Y 230.027,Z 605.549,A -85,B 0,C 180,E1 -19801.641,E2 -19801.641} C_VEL
LIN {X 0,Y 228.644,Z 603.228,A -85,B 0,C 180,E1 -19802.477,E2 -19802.477} C_VEL
LIN {X 0,Y 228.346,Z 602.036,A -85,B 0,C 180,E1 -19802.756,E2 -19802.756} C_VEL
LIN {X 0,Y 228.349,Z 602.03,A -85,B 0,C 180,E1 -19807.072,E2 -19807.072} C_VEL
LIN {X 0,Y 228.158,Z 602.05,A -85,B 0,C 180,E1 -19810.651,E2 -19810.651} C_VEL
LIN {X 0,Y 228.049,Z 602.065,A -85,B 0,C 180,E1 -19816.103,E2 -19816.103} C_VEL
LIN {X 0,Y 227.937,Z 602.08,A -85,B 0,C 180,E1 -19819.826,E2 -19819.826} C_VEL
LIN {X 0,Y 227.91,Z 602.085,A -85,B 0,C 180,E1 -19823.633,E2 -19823.633} C_VEL
LIN {X 0,Y 227.882,Z 602.09,A -85,B 0,C 180,E1 -19827.556,E2 -19827.556} C_VEL
LIN {X 0,Y 227.869,Z 602.096,A -85,B 0,C 180,E1 -19831.622,E2 -19831.622} C_VEL
LIN {X 0,Y 227.916,Z 602.196,A -85,B 0,C 180,E1 -19833.31,E2 -19833.31} C_VEL
LIN {X 0,Y 229.487,Z 606.816,A -85,B 0,C 180,E1 -19837.77,E2 -19837.77} C_VEL
LIN {X 0,Y 231.309,Z 612.179,A -85,B 0,C 180,E1 -19841.947,E2 -19841.947} C_VEL
LIN {X 0,Y 232.854,Z 617.122,A -85,B 0,C 180,E1 -19845.06,E2 -19845.06} C_VEL
LIN {X 0,Y 236.227,Z 622.704,A -85,B 0,C 180,E1 -19846.718,E2 -19846.718} C_VEL
LIN {X 0,Y 237.595,Z 624.904,A -85,B 0,C 180,E1 -19847.344,E2 -19847.344} C_VEL
LIN {X 0,Y 241.217,Z 631.31,A -85,B 0,C 180,E1 -19848.928,E2 -19848.928} C_VEL
LIN {X 0,Y 244.705,Z 637.862,A -85,B 0,C 180,E1 -19850.346,E2 -19850.346} C_VEL
LIN {X 0,Y 248.806,Z 646.342,A -85,B 0,C 180,E1 -19851.929,E2 -19851.929} C_VEL
LIN {X 0,Y 252.724,Z 655.785,A -85,B 0,C 180,E1 -19853.382,E2 -19853.382} C_VEL
LIN {X 0,Y 254.875,Z 675.251,A -85,B 0,C 180,E1 -19854.824,E2 -19854.824} C_VEL
LIN {X 0,Y 255.795,Z 692.91,A -85,B 0,C 180,E1 -19855.852,E2 -19855.852} C_VEL
LIN {X 0,Y 253.162,Z 732.348,A -85,B 0,C 180,E1 -19857.172,E2 -19857.172} C_VEL
LIN {X 0,Y 251.383,Z 746.305,A -85,B 0,C 180,E1 -19857.915,E2 -19857.915} C_VEL
LIN {X 0,Y 249.25,Z 758.004,A -85,B 0,C 180,E1 -19858.795,E2 -19858.795} C_VEL
LIN {X 0,Y 246.385,Z 770.419,A -85,B 0,C 180,E1 -19860.055,E2 -19860.055} C_VEL
LIN {X 0,Y 243.394,Z 781.643,A -85,B 0,C 180,E1 -19861.548,E2 -19861.548} C_VEL
LIN {X 0,Y 240.252,Z 791.921,A -85,B 0,C 180,E1 -19863.273,E2 -19863.273} C_VEL
LIN {X 0,Y 236.921,Z 802.13,A -85,B 0,C 180,E1 -19865.463,E2 -19865.463} C_VEL
LIN {X 0,Y 233.747,Z 811.224,A -85,B 0,C 180,E1 -19867.925,E2 -19867.925} C_VEL
LIN {X 0,Y 231.304,Z 818.606,A -85,B 0,C 180,E1 -19870.475,E2 -19870.475} C_VEL
LIN {X 0,Y 229.182,Z 824.576,A -85,B 0,C 180,E1 -19873.063,E2 -19873.063} C_VEL
LIN {X 0,Y 227.656,Z 829.366,A -85,B 0,C 180,E1 -19875.702,E2 -19875.702} C_VEL
LIN {X 0,Y 226.605,Z 833.109,A -85,B 0,C 180,E1 -19878.37,E2 -19878.37} C_VEL
LIN {X 0,Y 226.127,Z 835.865,A -85,B 0,C 180,E1 -19881.06,E2 -19881.06} C_VEL
LIN {X 0,Y 226.092,Z 838.049,A -85,B 0,C 180,E1 -19884.649,E2 -19884.649} C_VEL
LIN {X 0,Y 226.451,Z 838.641,A -85,B 0,C 180,E1 -19888.222,E2 -19888.222} C_VEL
LIN {X 0,Y 226.65,Z 838.278,A -85,B 0,C 180,E1 -19890,E2 -19890} C_VEL
LIN {X 0,Y 226.559,Z 837.452,A -85,B 0,C 180,E1 -19891.778,E2 -19891.778} C_VEL
LIN {X 0,Y 226.119,Z 837.032,A -85,B 0,C 180,E1 -19895.35,E2 -19895.35} C_VEL
LIN {X 0,Y 226.007,Z 836.235,A -85,B 0,C 180,E1 -19897.145,E2 -19897.145} C_VEL
LIN {X 0,Y 226.11,Z 835.031,A -85,B 0,C 180,E1 -19898.94,E2 -19898.94} C_VEL
LIN {X 0,Y 226.608,Z 832.442,A -85,B 0,C 180,E1 -19901.63,E2 -19901.63} C_VEL
LIN {X 0,Y 227.668,Z 828.871,A -85,B 0,C 180,E1 -19904.297,E2 -19904.297} C_VEL
LIN {X 0,Y 229.192,Z 824.217,A -85,B 0,C 180,E1 -19906.936,E2 -19906.936} C_VEL
LIN {X 0,Y 231.148,Z 818.335,A -85,B 0,C 180,E1 -19909.539,E2 -19909.539} C_VEL
LIN {X 0,Y 233.687,Z 811.037,A -85,B 0,C 180,E1 -19912.081,E2 -19912.081} C_VEL
LIN {X 0,Y 236.877,Z 802.03,A -85,B 0,C 180,E1 -19914.542,E2 -19914.542} C_VEL
LIN {X 0,Y 239.946,Z 792.733,A -85,B 0,C 180,E1 -19916.53,E2 -19916.53} C_VEL
LIN {X 0,Y 242.934,Z 782.434,A -85,B 0,C 180,E1 -19918.275,E2 -19918.275} C_VEL
LIN {X 0,Y 245.554,Z 772.585,A -85,B 0,C 180,E1 -19919.584,E2 -19919.584} C_VEL
LIN {X 0,Y 248.28,Z 760.114,A -85,B 0,C 180,E1 -19920.867,E2 -19920.867} C_VEL
LIN {X 0,Y 250.485,Z 747.238,A -85,B 0,C 180,E1 -19921.799,E2 -19921.799} C_VEL
LIN {X 0,Y 251.94,Z 734.075,A -85,B 0,C 180,E1 -19922.454,E2 -19922.454} C_VEL
LIN {X 0,Y 254.143,Z 688.715,A -85,B 0,C 180,E1 -19923.742,E2 -19923.742} C_VEL
LIN {X 0,Y 252.329,Z 665.329,A -85,B 0,C 180,E1 -19924.91,E2 -19924.91} C_VEL
LIN {X 0,Y 250.509,Z 649.354,A -85,B 0,C 180,E1 -19925.841,E2 -19925.841} C_VEL
LIN {X 0,Y 244.426,Z 633.718,A -85,B 0,C 180,E1 -19927.66,E2 -19927.66} C_VEL
LIN {X 0,Y 238.698,Z 620.152,A -85,B 0,C 180,E1 -19929.469,E2 -19929.469} C_VEL
LIN {X 0,Y 236.306,Z 616.366,A -85,B 0,C 180,E1 -19930.191,E2 -19930.191} C_VEL
LIN {X 0,Y 232.816,Z 610.876,A -85,B 0,C 180,E1 -19931.338,E2 -19931.338} C_VEL
LIN {X 0,Y 229.6,Z 605.903,A -85,B 0,C 180,E1 -19932.723,E2 -19932.723} C_VEL
LIN {X 0,Y 228.309,Z 603.735,A -85,B 0,C 180,E1 -19933.326,E2 -19933.326} C_VEL
LIN {X 0,Y 227.905,Z 602.097,A -85,B 0,C 180,E1 -19933.638,E2 -19933.638} C_VEL
LIN {X 0,Y 227.907,Z 602.096,A -85,B 0,C 180,E1 -19937.737,E2 -19937.737} C_VEL
LIN {X 0,Y 227.869,Z 602.095,A -85,B 0,C 180,E1 -19941.914,E2 -19941.914} C_VEL
LIN {X 0,Y 227.887,Z 602.082,A -85,B 0,C 180,E1 -19946.372,E2 -19946.372} C_VEL
LIN {X 0,Y 227.901,Z 602.075,A -85,B 0,C 180,E1 -19950.435,E2 -19950.435} C_VEL
LIN {X 0,Y 227.924,Z 602.094,A -85,B 0,C 180,E1 -19954.425,E2 -19954.425} C_VEL
LIN {X 0,Y 227.958,Z 602.067,A -85,B 0,C 180,E1 -19958.287,E2 -19958.287} C_VEL
LIN {X 0,Y 228.029,Z 602.06,A -85,B 0,C 180,E1 -19962.826,E2 -19962.826} C_VEL
LIN {X 0,Y 228.066,Z 602.076,A -85,B 0,C 180,E1 -19967.543,E2 -19967.543} C_VEL
LIN {X 0,Y 228.262,Z 602.022,A -85,B 0,C 180,E1 -19971.144,E2 -19971.144} C_VEL
LIN {X 0,Y 228.319,Z 602.028,A -85,B 0,C 180,E1 -19972.927,E2 -19972.927} C_VEL
LIN {X 0,Y 228.55,Z 601.986,A -85,B 0,C 180,E1 -19978.238,E2 -19978.238} C_VEL
LIN {X 0,Y 228.551,Z 602.015,A -85,B 0,C 180,E1 -19981.762,E2 -19981.762} C_VEL
LIN {X 0,Y 228.348,Z 602.02,A -85,B 0,C 180,E1 -19987.072,E2 -19987.072} C_VEL
LIN {X 0,Y 228.154,Z 602.054,A -85,B 0,C 180,E1 -19990.651,E2 -19990.651} C_VEL
LIN {X 0,Y 228.059,Z 602.065,A -85,B 0,C 180,E1 -19994.272,E2 -19994.272} C_VEL
LIN {X 0,Y 227.998,Z 602.066,A -85,B 0,C 180,E1 -19997.954,E2 -19997.954} C_VEL
LIN {X 0,Y 227.926,Z 602.094,A -85,B 0,C 180,E1 -20002.33,E2 -20002.33} C_VEL
LIN {X 0,Y 227.939,Z 602.088,A -85,B 0,C 180,E1 -20006.603,E2 -20006.603} C_VEL
LIN {X 0,Y 227.905,Z 602.08,A -85,B 0,C 180,E1 -20010.297,E2 -20010.297} C_VEL
LIN {X 0,Y 227.886,Z 602.087,A -85,B 0,C 180,E1 -20013.719,E2 -20013.719} C_VEL
LIN {X 0,Y 227.919,Z 602.142,A -85,B 0,C 180,E1 -20015.993,E2 -20015.993} C_VEL
LIN {X 0,Y 228.865,Z 604.832,A -85,B 0,C 180,E1 -20016.373,E2 -20016.373} C_VEL
LIN {X 0,Y 231.292,Z 607.658,A -85,B 0,C 180,E1 -20017.142,E2 -20017.142} C_VEL
LIN {X 0,Y 233.491,Z 610.987,A -85,B 0,C 180,E1 -20017.849,E2 -20017.849} C_VEL
LIN {X 0,Y 240.109,Z 620.604,A -85,B 0,C 180,E1 -20019.83,E2 -20019.83} C_VEL
LIN {X 0,Y 248.294,Z 633.949,A -85,B 0,C 180,E1 -20022.104,E2 -20022.104} C_VEL
LIN {X 0,Y 255.354,Z 646.892,A -85,B 0,C 180,E1 -20023.939,E2 -20023.939} C_VEL
LIN {X 0,Y 256.294,Z 648.783,A -85,B 0,C 180,E1 -20024.178,E2 -20024.178} C_VEL
LIN {X 0,Y 254.335,Z 691.935,A -85,B 0,C 180,E1 -20025.361,E2 -20025.361} C_VEL
LIN {X 0,Y 253.523,Z 705.353,A -85,B 0,C 180,E1 -20025.928,E2 -20025.928} C_VEL
LIN {X 0,Y 252.207,Z 717.832,A -85,B 0,C 180,E1 -20026.769,E2 -20026.769} C_VEL
LIN {X 0,Y 250.26,Z 730.155,A -85,B 0,C 180,E1 -20027.897,E2 -20027.897} C_VEL
LIN {X 0,Y 247.953,Z 741.657,A -85,B 0,C 180,E1 -20029.315,E2 -20029.315} C_VEL
LIN {X 0,Y 245.039,Z 753.199,A -85,B 0,C 180,E1 -20031.143,E2 -20031.143} C_VEL
LIN {X 0,Y 242.287,Z 762.425,A -85,B 0,C 180,E1 -20032.995,E2 -20032.995} C_VEL
LIN {X 0,Y 239.235,Z 771.592,A -85,B 0,C 180,E1 -20035.342,E2 -20035.342} C_VEL
LIN {X 0,Y 236.586,Z 778.825,A -85,B 0,C 180,E1 -20037.677,E2 -20037.677} C_VEL
LIN {X 0,Y 234.022,Z 785.107,A -85,B 0,C 180,E1 -20040.231,E2 -20040.231} C_VEL
LIN {X 0,Y 231.81,Z 790.213,A -85,B 0,C 180,E1 -20042.951,E2 -20042.951} C_VEL
LIN {X 0,Y 230.025,Z 793.992,A -85,B 0,C 180,E1 -20045.641,E2 -20045.641} C_VEL
LIN {X 0,Y 228.632,Z 796.692,A -85,B 0,C 180,E1 -20048.354,E2 -20048.354} C_VEL
LIN {X 0,Y 227.875,Z 797.934,A -85,B 0,C 180,E1 -20050.169,E2 -20050.169} C_VEL
LIN {X 0,Y 227.291,Z 798.771,A -85,B 0,C 180,E1 -20051.989,E2 -20051.989} C_VEL
LIN {X 0,Y 226.903,Z 799.151,A -85,B 0,C 180,E1 -20053.814,E2 -20053.814} C_VEL
LIN {X 0,Y 226.606,Z 799.13,A -85,B 0,C 180,E1 -20055.634,E2 -20055.634} C_VEL
LIN {X 0,Y 226.381,Z 798.727,A -85,B 0,C 180,E1 -20057.449,E2 -20057.449} C_VEL
LIN {X 0,Y 226.376,Z 797.901,A -85,B 0,C 180,E1 -20059.265,E2 -20059.265} C_VEL
LIN {X 0,Y 226.667,Z 795.029,A -85,B 0,C 180,E1 -20062.835,E2 -20062.835} C_VEL
LIN {X 0,Y 227.185,Z 791.671,A -85,B 0,C 180,E1 -20065.565,E2 -20065.565} C_VEL
LIN {X 0,Y 227.885,Z 787.298,A -85,B 0,C 180,E1 -20068.233,E2 -20068.233} C_VEL
LIN {X 0,Y 229.159,Z 780.641,A -85,B 0,C 180,E1 -20071.318,E2 -20071.318} C_VEL
LIN {X 0,Y 230.528,Z 773.409,A -85,B 0,C 180,E1 -20073.933,E2 -20073.933} C_VEL
LIN {X 0,Y 232.028,Z 766.015,A -85,B 0,C 180,E1 -20076.085,E2 -20076.085} C_VEL
LIN {X 0,Y 233.725,Z 757.078,A -85,B 0,C 180,E1 -20078.211,E2 -20078.211} C_VEL
LIN {X 0,Y 235.346,Z 747.195,A -85,B 0,C 180,E1 -20080.104,E2 -20080.104} C_VEL
LIN {X 0,Y 237.026,Z 736.416,A -85,B 0,C 180,E1 -20081.74,E2 -20081.74} C_VEL
LIN {X 0,Y 238.569,Z 724.318,A -85,B 0,C 180,E1 -20083.168,E2 -20083.168} C_VEL
LIN {X 0,Y 239.745,Z 711.57,A -85,B 0,C 180,E1 -20084.271,E2 -20084.271} C_VEL
LIN {X 0,Y 240.522,Z 698.206,A -85,B 0,C 180,E1 -20085.068,E2 -20085.068} C_VEL
LIN {X 0,Y 241.345,Z 672.141,A -85,B 0,C 180,E1 -20085.894,E2 -20085.894} C_VEL
LIN {X 0,Y 242.464,Z 635.871,A -85,B 0,C 180,E1 -20086.955,E2 -20086.955} C_VEL
LIN {X 0,Y 242.891,Z 637.446,A -85,B 0,C 180,E1 -20087.055,E2 -20087.055} C_VEL
LIN {X 0,Y 240.485,Z 695.275,A -85,B 0,C 180,E1 -20089.001,E2 -20089.001} C_VEL
LIN {X 0,Y 239.83,Z 707.635,A -85,B 0,C 180,E1 -20089.708,E2 -20089.708} C_VEL
LIN {X 0,Y 238.564,Z 721.186,A -85,B 0,C 180,E1 -20090.815,E2 -20090.815} C_VEL
LIN {X 0,Y 237.102,Z 733.539,A -85,B 0,C 180,E1 -20092.205,E2 -20092.205} C_VEL
LIN {X 0,Y 235.376,Z 745.86,A -85,B 0,C 180,E1 -20094.011,E2 -20094.011} C_VEL
LIN {X 0,Y 233.719,Z 755.741,A -85,B 0,C 180,E1 -20095.835,E2 -20095.835} C_VEL
LIN {X 0,Y 232.083,Z 765.093,A -85,B 0,C 180,E1 -20097.983,E2 -20097.983} C_VEL
LIN {X 0,Y 230.34,Z 774.419,A -85,B 0,C 180,E1 -20100.647,E2 -20100.647} C_VEL
LIN {X 0,Y 229.087,Z 780.988,A -85,B 0,C 180,E1 -20102.992,E2 -20102.992} C_VEL
LIN {X 0,Y 227.959,Z 787.354,A -85,B 0,C 180,E1 -20105.857,E2 -20105.857} C_VEL
LIN {X 0,Y 227.304,Z 791.479,A -85,B 0,C 180,E1 -20108.197,E2 -20108.197} C_VEL
LIN {X 0,Y 226.711,Z 794.823,A -85,B 0,C 180,E1 -20110.615,E2 -20110.615} C_VEL
LIN {X 0,Y 226.381,Z 797.331,A -85,B 0,C 180,E1 -20113.076,E2 -20113.076} C_VEL
LIN {X 0,Y 226.305,Z 799.059,A -85,B 0,C 180,E1 -20115.582,E2 -20115.582} C_VEL
LIN {X 0,Y 226.458,Z 800.003,A -85,B 0,C 180,E1 -20118.142,E2 -20118.142} C_VEL
LIN {X 0,Y 227.242,Z 799.912,A -85,B 0,C 180,E1 -20121.79,E2 -20121.79} C_VEL
LIN {X 0,Y 228.078,Z 798.901,A -85,B 0,C 180,E1 -20124.164,E2 -20124.164} C_VEL
LIN {X 0,Y 229.094,Z 797.223,A -85,B 0,C 180,E1 -20126.482,E2 -20126.482} C_VEL
LIN {X 0,Y 230.361,Z 794.844,A -85,B 0,C 180,E1 -20128.758,E2 -20128.758} C_VEL
LIN {X 0,Y 232.157,Z 791.063,A -85,B 0,C 180,E1 -20131.388,E2 -20131.388} C_VEL
LIN {X 0,Y 234.417,Z 785.892,A -85,B 0,C 180,E1 -20134.08,E2 -20134.08} C_VEL
LIN {X 0,Y 237.146,Z 779.211,A -85,B 0,C 180,E1 -20136.734,E2 -20136.734} C_VEL
LIN {X 0,Y 240.322,Z 770.737,A -85,B 0,C 180,E1 -20139.355,E2 -20139.355} C_VEL
LIN {X 0,Y 243.237,Z 762.003,A -85,B 0,C 180,E1 -20141.468,E2 -20141.468} C_VEL
LIN {X 0,Y 246.123,Z 751.993,A -85,B 0,C 180,E1 -20143.408,E2 -20143.408} C_VEL
LIN {X 0,Y 248.828,Z 741.368,A -85,B 0,C 180,E1 -20145.03,E2 -20145.03} C_VEL
LIN {X 0,Y 251.201,Z 729.471,A -85,B 0,C 180,E1 -20146.45,E2 -20146.45} C_VEL
LIN {X 0,Y 253.118,Z 717.305,A -85,B 0,C 180,E1 -20147.546,E2 -20147.546} C_VEL
LIN {X 0,Y 254.422,Z 705.037,A -85,B 0,C 180,E1 -20148.365,E2 -20148.365} C_VEL
LIN {X 0,Y 255.382,Z 691.133,A -85,B 0,C 180,E1 -20148.95,E2 -20148.95} C_VEL
LIN {X 0,Y 257.188,Z 663.661,A -85,B 0,C 180,E1 -20149.852,E2 -20149.852} C_VEL
LIN {X 0,Y 256.917,Z 659.906,A -85,B 0,C 180,E1 -20150.091,E2 -20150.091} C_VEL
LIN {X 0,Y 255.889,Z 656.5,A -85,B 0,C 180,E1 -20150.485,E2 -20150.485} C_VEL
LIN {X 0,Y 250.53,Z 646.449,A -85,B 0,C 180,E1 -20152.252,E2 -20152.252} C_VEL
LIN {X 0,Y 243.648,Z 634.122,A -85,B 0,C 180,E1 -20154.796,E2 -20154.796} C_VEL
LIN {X 0,Y 239.312,Z 627.384,A -85,B 0,C 180,E1 -20156.562,E2 -20156.562} C_VEL
LIN {X 0,Y 235.461,Z 622.084,A -85,B 0,C 180,E1 -20158.231,E2 -20158.231} C_VEL
LIN {X 0,Y 232.698,Z 617.904,A -85,B 0,C 180,E1 -20159.581,E2 -20159.581} C_VEL
LIN {X 0,Y 230.384,Z 614.704,A -85,B 0,C 180,E1 -20160.76,E2 -20160.76} C_VEL
LIN {X 0,Y 229.714,Z 613.705,A -85,B 0,C 180,E1 -20161.127,E2 -20161.127} C_VEL
LIN {X 0,Y 227.018,Z 610.968,A -85,B 0,C 180,E1 -20162.606,E2 -20162.606} C_VEL
LIN {X 0,Y 225.693,Z 608.663,A -85,B 0,C 180,E1 -20163.459,E2 -20163.459} C_VEL
LIN {X 0,Y 222.998,Z 606.913,A -85,B 0,C 180,E1 -20165.085,E2 -20165.085} C_VEL
LIN {X 0,Y 221.626,Z 604.599,A -85,B 0,C 180,E1 -20166.144,E2 -20166.144} C_VEL
LIN {X 0,Y 221.251,Z 602.914,A -85,B 0,C 180,E1 -20166.612,E2 -20166.612} C_VEL
LIN {X 0,Y 221.184,Z 602.919,A -85,B 0,C 180,E1 -20169.942,E2 -20169.942} C_VEL
LIN {X 0,Y 220.987,Z 602.945,A -85,B 0,C 180,E1 -20174.739,E2 -20174.739} C_VEL
LIN {X 0,Y 220.917,Z 602.959,A -85,B 0,C 180,E1 -20178.55,E2 -20178.55} C_VEL
LIN {X 0,Y 220.892,Z 602.965,A -85,B 0,C 180,E1 -20182.683,E2 -20182.683} C_VEL
LIN {X 0,Y 220.882,Z 602.962,A -85,B 0,C 180,E1 -20187.016,E2 -20187.016} C_VEL
LIN {X 0,Y 220.87,Z 603.117,A -85,B 0,C 180,E1 -20189.29,E2 -20189.29} C_VEL
LIN {X 0,Y 221.753,Z 605.58,A -85,B 0,C 180,E1 -20192.601,E2 -20192.601} C_VEL
LIN {X 0,Y 223.109,Z 609.578,A -85,B 0,C 180,E1 -20196.763,E2 -20196.763} C_VEL
LIN {X 0,Y 224.385,Z 613.272,A -85,B 0,C 180,E1 -20199.948,E2 -20199.948} C_VEL
LIN {X 0,Y 225.155,Z 615.418,A -85,B 0,C 180,E1 -20201.486,E2 -20201.486} C_VEL
LIN {X 0,Y 228.78,Z 621.351,A -85,B 0,C 180,E1 -20203.685,E2 -20203.685} C_VEL
LIN {X 0,Y 230.182,Z 623.394,A -85,B 0,C 180,E1 -20204.435,E2 -20204.435} C_VEL
LIN {X 0,Y 233.796,Z 629.213,A -85,B 0,C 180,E1 -20206.277,E2 -20206.277} C_VEL
LIN {X 0,Y 237.847,Z 636.754,A -85,B 0,C 180,E1 -20208.174,E2 -20208.174} C_VEL
LIN {X 0,Y 240.979,Z 642.869,A -85,B 0,C 180,E1 -20209.547,E2 -20209.547} C_VEL
LIN {X 0,Y 245.03,Z 651.62,A -85,B 0,C 180,E1 -20211.199,E2 -20211.199} C_VEL
LIN {X 0,Y 247.951,Z 658.78,A -85,B 0,C 180,E1 -20212.368,E2 -20212.368} C_VEL
LIN {X 0,Y 249.769,Z 676.208,A -85,B 0,C 180,E1 -20213.703,E2 -20213.703} C_VEL
LIN {X 0,Y 250.651,Z 693.508,A -85,B 0,C 180,E1 -20214.759,E2 -20214.759} C_VEL
LIN {X 0,Y 247.921,Z 731.446,A -85,B 0,C 180,E1 -20216.051,E2 -20216.051} C_VEL
LIN {X 0,Y 246.151,Z 745.232,A -85,B 0,C 180,E1 -20216.807,E2 -20216.807} C_VEL
LIN {X 0,Y 243.715,Z 757.817,A -85,B 0,C 180,E1 -20217.76,E2 -20217.76} C_VEL
LIN {X 0,Y 240.732,Z 770.132,A -85,B 0,C 180,E1 -20219.034,E2 -20219.034} C_VEL
LIN {X 0,Y 237.61,Z 781.292,A -85,B 0,C 180,E1 -20220.546,E2 -20220.546} C_VEL
LIN {X 0,Y 234.331,Z 791.502,A -85,B 0,C 180,E1 -20222.299,E2 -20222.299} C_VEL
LIN {X 0,Y 231.106,Z 800.799,A -85,B 0,C 180,E1 -20224.321,E2 -20224.321} C_VEL
LIN {X 0,Y 227.695,Z 809.954,A -85,B 0,C 180,E1 -20226.826,E2 -20226.826} C_VEL
LIN {X 0,Y 224.931,Z 817.557,A -85,B 0,C 180,E1 -20229.469,E2 -20229.469} C_VEL
LIN {X 0,Y 223.136,Z 822.574,A -85,B 0,C 180,E1 -20231.642,E2 -20231.642} C_VEL
LIN {X 0,Y 221.232,Z 827.638,A -85,B 0,C 180,E1 -20234.335,E2 -20234.335} C_VEL
LIN {X 0,Y 219.869,Z 831.604,A -85,B 0,C 180,E1 -20237.071,E2 -20237.071} C_VEL
LIN {X 0,Y 219.373,Z 833.716,A -85,B 0,C 180,E1 -20238.918,E2 -20238.918} C_VEL
LIN {X 0,Y 219.062,Z 835.376,A -85,B 0,C 180,E1 -20240.769,E2 -20240.769} C_VEL
LIN {X 0,Y 219.015,Z 837.476,A -85,B 0,C 180,E1 -20244.476,E2 -20244.476} C_VEL
LIN {X 0,Y 219.094,Z 837.929,A -85,B 0,C 180,E1 -20246.322,E2 -20246.322} C_VEL
LIN {X 0,Y 219.376,Z 837.962,A -85,B 0,C 180,E1 -20248.164,E2 -20248.164} C_VEL
LIN {X 0,Y 219.595,Z 837.544,A -85,B 0,C 180,E1 -20250,E2 -20250} C_VEL
LIN {X 0,Y 219.474,Z 836.821,A -85,B 0,C 180,E1 -20251.835,E2 -20251.835} C_VEL
LIN {X 0,Y 219.043,Z 836.463,A -85,B 0,C 180,E1 -20255.523,E2 -20255.523} C_VEL
LIN {X 0,Y 219.049,Z 834.529,A -85,B 0,C 180,E1 -20259.231,E2 -20259.231} C_VEL
LIN {X 0,Y 219.614,Z 831.984,A -85,B 0,C 180,E1 -20262.005,E2 -20262.005} C_VEL
LIN {X 0,Y 220.74,Z 828.464,A -85,B 0,C 180,E1 -20264.756,E2 -20264.756} C_VEL
LIN {X 0,Y 222.386,Z 823.877,A -85,B 0,C 180,E1 -20267.471,E2 -20267.471} C_VEL
LIN {X 0,Y 224.431,Z 818.085,A -85,B 0,C 180,E1 -20270.148,E2 -20270.148} C_VEL
LIN {X 0,Y 227.111,Z 810.872,A -85,B 0,C 180,E1 -20272.756,E2 -20272.756} C_VEL
LIN {X 0,Y 230.433,Z 801.961,A -85,B 0,C 180,E1 -20275.276,E2 -20275.276} C_VEL
LIN {X 0,Y 233.638,Z 792.827,A -85,B 0,C 180,E1 -20277.305,E2 -20277.305} C_VEL
LIN {X 0,Y 236.725,Z 782.687,A -85,B 0,C 180,E1 -20279.087,E2 -20279.087} C_VEL
LIN {X 0,Y 239.811,Z 771.476,A -85,B 0,C 180,E1 -20280.61,E2 -20280.61} C_VEL
LIN {X 0,Y 242.469,Z 759.873,A -85,B 0,C 180,E1 -20281.813,E2 -20281.813} C_VEL
LIN {X 0,Y 244.738,Z 747.168,A -85,B 0,C 180,E1 -20282.759,E2 -20282.759} C_VEL
LIN {X 0,Y 246.234,Z 734.326,A -85,B 0,C 180,E1 -20283.422,E2 -20283.422} C_VEL
LIN {X 0,Y 247.669,Z 707.939,A -85,B 0,C 180,E1 -20284.213,E2 -20284.213} C_VEL
LIN {X 0,Y 248.5,Z 688.326,A -85,B 0,C 180,E1 -20284.781,E2 -20284.781} C_VEL
LIN {X 0,Y 246.693,Z 665.263,A -85,B 0,C 180,E1 -20285.988,E2 -20285.988} C_VEL
LIN {X 0,Y 245.223,Z 652.007,A -85,B 0,C 180,E1 -20286.788,E2 -20286.788} C_VEL
LIN {X 0,Y 239.214,Z 636.272,A -85,B 0,C 180,E1 -20288.691,E2 -20288.691} C_VEL
LIN {X 0,Y 234.001,Z 623.809,A -85,B 0,C 180,E1 -20290.432,E2 -20290.432} C_VEL
LIN {X 0,Y 227.444,Z 614.163,A -85,B 0,C 180,E1 -20292.543,E2 -20292.543} C_VEL
LIN {X 0,Y 224.844,Z 610.487,A -85,B 0,C 180,E1 -20293.444,E2 -20293.444} C_VEL
LIN {X 0,Y 223.036,Z 607.275,A -85,B 0,C 180,E1 -20294.361,E2 -20294.361} C_VEL
LIN {X 0,Y 221.296,Z 604.773,A -85,B 0,C 180,E1 -20295.195,E2 -20295.195} C_VEL
LIN {X 0,Y 220.81,Z 602.967,A -85,B 0,C 180,E1 -20295.607,E2 -20295.607} C_VEL
LIN {X 0,Y 220.85,Z 602.96,A -85,B 0,C 180,E1 -20299.793,E2 -20299.793} C_VEL
LIN {X 0,Y 220.833,Z 602.977,A -85,B 0,C 180,E1 -20302.794,E2 -20302.794} C_VEL
LIN {X 0,Y 220.82,Z 602.972,A -85,B 0,C 180,E1 -20307.244,E2 -20307.244} C_VEL
LIN {X 0,Y 220.823,Z 602.955,A -85,B 0,C 180,E1 -20311.484,E2 -20311.484} C_VEL
LIN {X 0,Y 220.863,Z 602.96,A -85,B 0,C 180,E1 -20315.564,E2 -20315.564} C_VEL
LIN {X 0,Y 220.888,Z 602.963,A -85,B 0,C 180,E1 -20319.513,E2 -20319.513} C_VEL
LIN {X 0,Y 221.01,Z 602.929,A -85,B 0,C 180,E1 -20323.37,E2 -20323.37} C_VEL
LIN {X 0,Y 221.062,Z 602.937,A -85,B 0,C 180,E1 -20329.003,E2 -20329.003} C_VEL
LIN {X 0,Y 221.255,Z 602.905,A -85,B 0,C 180,E1 -20332.7,E2 -20332.7} C_VEL
LIN {X 0,Y 221.508,Z 602.863,A -85,B 0,C 180,E1 -20338.182,E2 -20338.182} C_VEL
LIN {X 0,Y 221.509,Z 602.893,A -85,B 0,C 180,E1 -20341.818,E2 -20341.818} C_VEL
LIN {X 0,Y 221.283,Z 602.902,A -85,B 0,C 180,E1 -20347.299,E2 -20347.299} C_VEL
LIN {X 0,Y 221.102,Z 602.927,A -85,B 0,C 180,E1 -20350.995,E2 -20350.995} C_VEL
LIN {X 0,Y 221.012,Z 602.95,A -85,B 0,C 180,E1 -20356.63,E2 -20356.63} C_VEL
LIN {X 0,Y 220.888,Z 602.958,A -85,B 0,C 180,E1 -20360.487,E2 -20360.487} C_VEL
LIN {X 0,Y 220.863,Z 602.954,A -85,B 0,C 180,E1 -20364.436,E2 -20364.436} C_VEL
LIN {X 0,Y 220.833,Z 602.968,A -85,B 0,C 180,E1 -20368.514,E2 -20368.514} C_VEL
LIN {X 0,Y 220.821,Z 602.976,A -85,B 0,C 180,E1 -20372.755,E2 -20372.755} C_VEL
LIN {X 0,Y 220.863,Z 603.09,A -85,B 0,C 180,E1 -20373.998,E2 -20373.998} C_VEL
LIN {X 0,Y 221.711,Z 605.626,A -85,B 0,C 180,E1 -20374.378,E2 -20374.378} C_VEL
LIN {X 0,Y 223.805,Z 607.907,A -85,B 0,C 180,E1 -20375.104,E2 -20375.104} C_VEL
LIN {X 0,Y 224.452,Z 608.765,A -85,B 0,C 180,E1 -20375.33,E2 -20375.33} C_VEL
LIN {X 0,Y 226.648,Z 611.999,A -85,B 0,C 180,E1 -20376.098,E2 -20376.098} C_VEL
LIN {X 0,Y 227.877,Z 613.565,A -85,B 0,C 180,E1 -20376.505,E2 -20376.505} C_VEL
LIN {X 0,Y 235.935,Z 625.389,A -85,B 0,C 180,E1 -20379.059,E2 -20379.059} C_VEL
LIN {X 0,Y 243.899,Z 638.567,A -85,B 0,C 180,E1 -20381.376,E2 -20381.376} C_VEL
LIN {X 0,Y 250.704,Z 651.239,A -85,B 0,C 180,E1 -20383.224,E2 -20383.224} C_VEL
LIN {X 0,Y 248.886,Z 689.665,A -85,B 0,C 180,E1 -20384.292,E2 -20384.292} C_VEL
LIN {X 0,Y 248.117,Z 703.427,A -85,B 0,C 180,E1 -20384.825,E2 -20384.825} C_VEL
LIN {X 0,Y 246.912,Z 715.54,A -85,B 0,C 180,E1 -20385.578,E2 -20385.578} C_VEL
LIN {X 0,Y 245.237,Z 726.782,A -85,B 0,C 180,E1 -20386.546,E2 -20386.546} C_VEL
LIN {X 0,Y 242.753,Z 739.203,A -85,B 0,C 180,E1 -20387.973,E2 -20387.973} C_VEL
LIN {X 0,Y 240.246,Z 749.559,A -85,B 0,C 180,E1 -20389.516,E2 -20389.516} C_VEL
LIN {X 0,Y 237.436,Z 759.132,A -85,B 0,C 180,E1 -20391.298,E2 -20391.298} C_VEL
LIN {X 0,Y 234.721,Z 767.378,A -85,B 0,C 180,E1 -20393.214,E2 -20393.214} C_VEL
LIN {X 0,Y 231.955,Z 774.923,A -85,B 0,C 180,E1 -20395.383,E2 -20395.383} C_VEL
LIN {X 0,Y 228.984,Z 782.256,A -85,B 0,C 180,E1 -20398.033,E2 -20398.033} C_VEL
LIN {X 0,Y 226.799,Z 787.169,A -85,B 0,C 180,E1 -20400.278,E2 -20400.278} C_VEL
LIN {X 0,Y 224.631,Z 791.86,A -85,B 0,C 180,E1 -20403.022,E2 -20403.022} C_VEL
LIN {X 0,Y 222.575,Z 795.894,A -85,B 0,C 180,E1 -20406.306,E2 -20406.306} C_VEL
LIN {X 0,Y 221.024,Z 798.405,A -85,B 0,C 180,E1 -20409.527,E2 -20409.527} C_VEL
LIN {X 0,Y 220.38,Z 799.284,A -85,B 0,C 180,E1 -20411.404,E2 -20411.404} C_VEL
LIN {X 0,Y 219.901,Z 799.757,A -85,B 0,C 180,E1 -20413.496,E2 -20413.496} C_VEL
LIN {X 0,Y 219.336,Z 799.401,A -85,B 0,C 180,E1 -20417.039,E2 -20417.039} C_VEL
LIN {X 0,Y 219.293,Z 798.642,A -85,B 0,C 180,E1 -20418.914,E2 -20418.914} C_VEL
LIN {X 0,Y 219.363,Z 797.439,A -85,B 0,C 180,E1 -20420.782,E2 -20420.782} C_VEL
LIN {X 0,Y 219.58,Z 795.633,A -85,B 0,C 180,E1 -20422.841,E2 -20422.841} C_VEL
LIN {X 0,Y 220.063,Z 792.592,A -85,B 0,C 180,E1 -20425.421,E2 -20425.421} C_VEL
LIN {X 0,Y 220.776,Z 788.309,A -85,B 0,C 180,E1 -20428.176,E2 -20428.176} C_VEL
LIN {X 0,Y 221.832,Z 782.843,A -85,B 0,C 180,E1 -20430.908,E2 -20430.908} C_VEL
LIN {X 0,Y 223.182,Z 776.015,A -85,B 0,C 180,E1 -20433.611,E2 -20433.611} C_VEL
LIN {X 0,Y 224.978,Z 767.433,A -85,B 0,C 180,E1 -20436.277,E2 -20436.277} C_VEL
LIN {X 0,Y 226.745,Z 758.653,A -85,B 0,C 180,E1 -20438.466,E2 -20438.466} C_VEL
LIN {X 0,Y 228.389,Z 749.059,A -85,B 0,C 180,E1 -20440.415,E2 -20440.415} C_VEL
LIN {X 0,Y 230.146,Z 738.414,A -85,B 0,C 180,E1 -20442.119,E2 -20442.119} C_VEL
LIN {X 0,Y 231.764,Z 726.443,A -85,B 0,C 180,E1 -20443.612,E2 -20443.612} C_VEL
LIN {X 0,Y 233.059,Z 714.116,A -85,B 0,C 180,E1 -20444.761,E2 -20444.761} C_VEL
LIN {X 0,Y 233.901,Z 701.245,A -85,B 0,C 180,E1 -20445.597,E2 -20445.597} C_VEL
LIN {X 0,Y 234.447,Z 686.527,A -85,B 0,C 180,E1 -20446.162,E2 -20446.162} C_VEL
LIN {X 0,Y 235.43,Z 657.055,A -85,B 0,C 180,E1 -20447.028,E2 -20447.028} C_VEL
LIN {X 0,Y 233.725,Z 697.763,A -85,B 0,C 180,E1 -20448.518,E2 -20448.518} C_VEL
LIN {X 0,Y 232.848,Z 711.607,A -85,B 0,C 180,E1 -20449.39,E2 -20449.39} C_VEL
LIN {X 0,Y 231.579,Z 723.978,A -85,B 0,C 180,E1 -20450.513,E2 -20450.513} C_VEL
LIN {X 0,Y 230.085,Z 736.046,A -85,B 0,C 180,E1 -20451.973,E2 -20451.973} C_VEL
LIN {X 0,Y 228.553,Z 746.408,A -85,B 0,C 180,E1 -20453.562,E2 -20453.562} C_VEL
LIN {X 0,Y 226.796,Z 756.436,A -85,B 0,C 180,E1 -20455.464,E2 -20455.464} C_VEL
LIN {X 0,Y 224.921,Z 766.81,A -85,B 0,C 180,E1 -20457.949,E2 -20457.949} C_VEL
LIN {X 0,Y 223.443,Z 774.459,A -85,B 0,C 180,E1 -20460.214,E2 -20460.214} C_VEL
LIN {X 0,Y 221.961,Z 782.031,A -85,B 0,C 180,E1 -20462.992,E2 -20462.992} C_VEL
LIN {X 0,Y 220.816,Z 788.443,A -85,B 0,C 180,E1 -20466.02,E2 -20466.02} C_VEL
LIN {X 0,Y 220.117,Z 792.574,A -85,B 0,C 180,E1 -20468.505,E2 -20468.505} C_VEL
LIN {X 0,Y 219.568,Z 795.822,A -85,B 0,C 180,E1 -20471.006,E2 -20471.006} C_VEL
LIN {X 0,Y 219.355,Z 797.371,A -85,B 0,C 180,E1 -20472.531,E2 -20472.531} C_VEL
LIN {X 0,Y 219.231,Z 799.362,A -85,B 0,C 180,E1 -20475.149,E2 -20475.149} C_VEL
LIN {X 0,Y 219.357,Z 800.481,A -85,B 0,C 180,E1 -20477.715,E2 -20477.715} C_VEL
LIN {X 0,Y 219.793,Z 800.81,A -85,B 0,C 180,E1 -20480.245,E2 -20480.245} C_VEL
LIN {X 0,Y 220.486,Z 800.379,A -85,B 0,C 180,E1 -20482.831,E2 -20482.831} C_VEL
LIN {X 0,Y 221.586,Z 799.044,A -85,B 0,C 180,E1 -20485.549,E2 -20485.549} C_VEL
LIN {X 0,Y 222.986,Z 796.716,A -85,B 0,C 180,E1 -20488.316,E2 -20488.316} C_VEL
LIN {X 0,Y 224.81,Z 793.29,A -85,B 0,C 180,E1 -20491.082,E2 -20491.082} C_VEL
LIN {X 0,Y 227.544,Z 787.585,A -85,B 0,C 180,E1 -20494.379,E2 -20494.379} C_VEL
LIN {X 0,Y 230.386,Z 781.241,A -85,B 0,C 180,E1 -20497.111,E2 -20497.111} C_VEL
LIN {X 0,Y 233.227,Z 774.244,A -85,B 0,C 180,E1 -20499.459,E2 -20499.459} C_VEL
LIN {X 0,Y 236.583,Z 764.991,A -85,B 0,C 180,E1 -20501.912,E2 -20501.912} C_VEL
LIN {X 0,Y 239.504,Z 755.98,A -85,B 0,C 180,E1 -20503.8,E2 -20503.8} C_VEL
LIN {X 0,Y 242.305,Z 745.798,A -85,B 0,C 180,E1 -20505.513,E2 -20505.513} C_VEL
LIN {X 0,Y 245.122,Z 733.637,A -85,B 0,C 180,E1 -20507.111,E2 -20507.111} C_VEL
LIN {X 0,Y 247.374,Z 721.148,A -85,B 0,C 180,E1 -20508.355,E2 -20508.355} C_VEL
LIN {X 0,Y 249.016,Z 707.861,A -85,B 0,C 180,E1 -20509.321,E2 -20509.321} C_VEL
LIN {X 0,Y 250.035,Z 694.873,A -85,B 0,C 180,E1 -20509.942,E2 -20509.942} C_VEL
LIN {X 0,Y 253.031,Z 651.567,A -85,B 0,C 180,E1 -20511.383,E2 -20511.383} C_VEL
LIN {X 0,Y 250.53,Z 646.449,A -85,B 0,C 180,E1 -20512.252,E2 -20512.252} C_VEL
LIN {X 0,Y 248.065,Z 642.59,A -85,B 0,C 180,E1 -20513.099,E2 -20513.099} C_VEL
LIN {X 0,Y 245.054,Z 639.703,A -85,B 0,C 180,E1 -20514.08,E2 -20514.08} C_VEL
LIN {X 0,Y 236.75,Z 633.512,A -85,B 0,C 180,E1 -20517.021,E2 -20517.021} C_VEL
LIN {X 0,Y 234.974,Z 631.536,A -85,B 0,C 180,E1 -20517.76,E2 -20517.76} C_VEL
LIN {X 0,Y 232.427,Z 627.766,A -85,B 0,C 180,E1 -20518.98,E2 -20518.98} C_VEL
LIN {X 0,Y 229.859,Z 623.841,A -85,B 0,C 180,E1 -20520.293,E2 -20520.293} C_VEL
LIN {X 0,Y 227.189,Z 619.974,A -85,B 0,C 180,E1 -20521.773,E2 -20521.773} C_VEL
LIN {X 0,Y 224.428,Z 616.827,A -85,B 0,C 180,E1 -20523.38,E2 -20523.38} C_VEL
LIN {X 0,Y 223.395,Z 615.233,A -85,B 0,C 180,E1 -20524.059,E2 -20524.059} C_VEL
LIN {X 0,Y 220.664,Z 613.008,A -85,B 0,C 180,E1 -20525.861,E2 -20525.861} C_VEL
LIN {X 0,Y 219.159,Z 610.071,A -85,B 0,C 180,E1 -20527.141,E2 -20527.141} C_VEL
LIN {X 0,Y 218.89,Z 609.596,A -85,B 0,C 180,E1 -20527.379,E2 -20527.379} C_VEL
LIN {X 0,Y 215.901,Z 607.66,A -85,B 0,C 180,E1 -20529.92,E2 -20529.92} C_VEL
LIN {X 0,Y 214.24,Z 604.977,A -85,B 0,C 180,E1 -20531.891,E2 -20531.891} C_VEL
LIN {X 0,Y 213.988,Z 603.818,A -85,B 0,C 180,E1 -20532.447,E2 -20532.447} C_VEL
LIN {X 0,Y 213.928,Z 603.821,A -85,B 0,C 180,E1 -20537.695,E2 -20537.695} C_VEL
LIN {X 0,Y 213.845,Z 603.98,A -85,B 0,C 180,E1 -20542.14,E2 -20542.14} C_VEL
LIN {X 0,Y 214.614,Z 606.386,A -85,B 0,C 180,E1 -20547.853,E2 -20547.853} C_VEL
LIN {X 0,Y 215.043,Z 607.207,A -85,B 0,C 180,E1 -20549.356,E2 -20549.356} C_VEL
LIN {X 0,Y 216.118,Z 610.415,A -85,B 0,C 180,E1 -20553.561,E2 -20553.561} C_VEL
LIN {X 0,Y 217.105,Z 613.193,A -85,B 0,C 180,E1 -20556.391,E2 -20556.391} C_VEL
LIN {X 0,Y 222.929,Z 621.999,A -85,B 0,C 180,E1 -20560.933,E2 -20560.933} C_VEL
LIN {X 0,Y 226.779,Z 628.181,A -85,B 0,C 180,E1 -20563.34,E2 -20563.34} C_VEL
LIN {X 0,Y 231.397,Z 636.165,A -85,B 0,C 180,E1 -20565.846,E2 -20565.846} C_VEL
LIN {X 0,Y 234.583,Z 642.305,A -85,B 0,C 180,E1 -20567.427,E2 -20567.427} C_VEL
LIN {X 0,Y 238.653,Z 650.562,A -85,B 0,C 180,E1 -20569.285,E2 -20569.285} C_VEL
LIN {X 0,Y 243,Z 661.124,A -85,B 0,C 180,E1 -20571.165,E2 -20571.165} C_VEL
LIN {X 0,Y 243.508,Z 662.989,A -85,B 0,C 180,E1 -20571.409,E2 -20571.409} C_VEL
LIN {X 0,Y 245.144,Z 682.095,A -85,B 0,C 180,E1 -20572.881,E2 -20572.881} C_VEL
LIN {X 0,Y 245.598,Z 694.344,A -85,B 0,C 180,E1 -20573.623,E2 -20573.623} C_VEL
LIN {X 0,Y 242.82,Z 730.883,A -85,B 0,C 180,E1 -20574.884,E2 -20574.884} C_VEL
LIN {X 0,Y 240.959,Z 744.742,A -85,B 0,C 180,E1 -20575.655,E2 -20575.655} C_VEL
LIN {X 0,Y 238.259,Z 757.885,A -85,B 0,C 180,E1 -20576.676,E2 -20576.676} C_VEL
LIN {X 0,Y 235.167,Z 769.984,A -85,B 0,C 180,E1 -20577.964,E2 -20577.964} C_VEL
LIN {X 0,Y 231.904,Z 780.989,A -85,B 0,C 180,E1 -20579.496,E2 -20579.496} C_VEL
LIN {X 0,Y 228.494,Z 791.075,A -85,B 0,C 180,E1 -20581.277,E2 -20581.277} C_VEL
LIN {X 0,Y 224.732,Z 801.171,A -85,B 0,C 180,E1 -20583.537,E2 -20583.537} C_VEL
LIN {X 0,Y 221.2,Z 810.164,A -85,B 0,C 180,E1 -20586.104,E2 -20586.104} C_VEL
LIN {X 0,Y 218.307,Z 817.441,A -85,B 0,C 180,E1 -20588.767,E2 -20588.767} C_VEL
LIN {X 0,Y 215.607,Z 824.211,A -85,B 0,C 180,E1 -20591.961,E2 -20591.961} C_VEL
LIN {X 0,Y 213.83,Z 828.789,A -85,B 0,C 180,E1 -20594.756,E2 -20594.756} C_VEL
LIN {X 0,Y 212.606,Z 832.323,A -85,B 0,C 180,E1 -20597.593,E2 -20597.593} C_VEL
LIN {X 0,Y 212.017,Z 834.897,A -85,B 0,C 180,E1 -20600.46,E2 -20600.46} C_VEL
LIN {X 0,Y 211.932,Z 836.906,A -85,B 0,C 180,E1 -20604.291,E2 -20604.291} C_VEL
LIN {X 0,Y 212.021,Z 837.304,A -85,B 0,C 180,E1 -20606.199,E2 -20606.199} C_VEL
LIN {X 0,Y 212.302,Z 837.268,A -85,B 0,C 180,E1 -20608.103,E2 -20608.103} C_VEL
LIN {X 0,Y 212.541,Z 836.811,A -85,B 0,C 180,E1 -20610,E2 -20610} C_VEL
LIN {X 0,Y 212.392,Z 836.184,A -85,B 0,C 180,E1 -20611.896,E2 -20611.896} C_VEL
LIN {X 0,Y 212.073,Z 836.245,A -85,B 0,C 180,E1 -20613.8,E2 -20613.8} C_VEL
LIN {X 0,Y 211.928,Z 835.862,A -85,B 0,C 180,E1 -20615.806,E2 -20615.806} C_VEL
LIN {X 0,Y 212.007,Z 834.015,A -85,B 0,C 180,E1 -20619.541,E2 -20619.541} C_VEL
LIN {X 0,Y 212.36,Z 832.455,A -85,B 0,C 180,E1 -20621.453,E2 -20621.453} C_VEL
LIN {X 0,Y 213.364,Z 829.333,A -85,B 0,C 180,E1 -20624.302,E2 -20624.302} C_VEL
LIN {X 0,Y 214.909,Z 825.177,A -85,B 0,C 180,E1 -20627.116,E2 -20627.116} C_VEL
LIN {X 0,Y 217.297,Z 818.957,A -85,B 0,C 180,E1 -20630.29,E2 -20630.29} C_VEL
LIN {X 0,Y 220.038,Z 811.999,A -85,B 0,C 180,E1 -20633.033,E2 -20633.033} C_VEL
LIN {X 0,Y 223.404,Z 803.516,A -85,B 0,C 180,E1 -20635.629,E2 -20635.629} C_VEL
LIN {X 0,Y 226.646,Z 794.816,A -85,B 0,C 180,E1 -20637.718,E2 -20637.718} C_VEL
LIN {X 0,Y 230.178,Z 784.14,A -85,B 0,C 180,E1 -20639.745,E2 -20639.745} C_VEL
LIN {X 0,Y 233.329,Z 773.481,A -85,B 0,C 180,E1 -20641.303,E2 -20641.303} C_VEL
LIN {X 0,Y 236.283,Z 761.564,A -85,B 0,C 180,E1 -20642.622,E2 -20642.622} C_VEL
LIN {X 0,Y 238.734,Z 749.192,A -85,B 0,C 180,E1 -20643.628,E2 -20643.628} C_VEL
LIN {X 0,Y 240.455,Z 736.195,A -85,B 0,C 180,E1 -20644.364,E2 -20644.364} C_VEL
LIN {X 0,Y 241.619,Z 720.036,A -85,B 0,C 180,E1 -20644.902,E2 -20644.902} C_VEL
LIN {X 0,Y 243.052,Z 690.096,A -85,B 0,C 180,E1 -20645.763,E2 -20645.763} C_VEL
LIN {X 0,Y 241.353,Z 667.074,A -85,B 0,C 180,E1 -20646.999,E2 -20646.999} C_VEL
LIN {X 0,Y 240.045,Z 654.67,A -85,B 0,C 180,E1 -20647.767,E2 -20647.767} C_VEL
LIN {X 0,Y 232.886,Z 635.725,A -85,B 0,C 180,E1 -20650.193,E2 -20650.193} C_VEL
LIN {X 0,Y 229.635,Z 628.248,A -85,B 0,C 180,E1 -20651.331,E2 -20651.331} C_VEL
LIN {X 0,Y 222.268,Z 617.15,A -85,B 0,C 180,E1 -20653.854,E2 -20653.854} C_VEL
LIN {X 0,Y 218.179,Z 611.651,A -85,B 0,C 180,E1 -20655.362,E2 -20655.362} C_VEL
LIN {X 0,Y 216.147,Z 608.3,A -85,B 0,C 180,E1 -20656.295,E2 -20656.295} C_VEL
LIN {X 0,Y 214.468,Z 606.033,A -85,B 0,C 180,E1 -20657.159,E2 -20657.159} C_VEL
LIN {X 0,Y 213.804,Z 603.853,A -85,B 0,C 180,E1 -20657.714,E2 -20657.714} C_VEL
LIN {X 0,Y 213.78,Z 603.851,A -85,B 0,C 180,E1 -20662.09,E2 -20662.09} C_VEL
LIN {X 0,Y 213.766,Z 603.838,A -85,B 0,C 180,E1 -20666.019,E2 -20666.019} C_VEL
LIN {X 0,Y 213.757,Z 603.836,A -85,B 0,C 180,E1 -20670.45,E2 -20670.45} C_VEL
LIN {X 0,Y 213.798,Z 603.852,A -85,B 0,C 180,E1 -20674.701,E2 -20674.701} C_VEL
LIN {X 0,Y 213.808,Z 603.833,A -85,B 0,C 180,E1 -20678.803,E2 -20678.803} C_VEL
LIN {X 0,Y 213.938,Z 603.814,A -85,B 0,C 180,E1 -20682.803,E2 -20682.803} C_VEL
LIN {X 0,Y 213.946,Z 603.83,A -85,B 0,C 180,E1 -20686.706,E2 -20686.706} C_VEL
LIN {X 0,Y 214.137,Z 603.782,A -85,B 0,C 180,E1 -20690.555,E2 -20690.555} C_VEL
LIN {X 0,Y 214.098,Z 603.815,A -85,B 0,C 180,E1 -20694.348,E2 -20694.348} C_VEL
LIN {X 0,Y 214.441,Z 603.743,A -85,B 0,C 180,E1 -20698.122,E2 -20698.122} C_VEL
LIN {X 0,Y 214.545,Z 603.739,A -85,B 0,C 180,E1 -20700,E2 -20700} C_VEL
LIN {X 0,Y 214.443,Z 603.773,A -85,B 0,C 180,E1 -20701.878,E2 -20701.878} C_VEL
LIN {X 0,Y 214.222,Z 603.785,A -85,B 0,C 180,E1 -20707.541,E2 -20707.541} C_VEL
LIN {X 0,Y 214.018,Z 603.805,A -85,B 0,C 180,E1 -20711.363,E2 -20711.363} C_VEL
LIN {X 0,Y 213.929,Z 603.835,A -85,B 0,C 180,E1 -20715.237,E2 -20715.237} C_VEL
LIN {X 0,Y 213.835,Z 603.826,A -85,B 0,C 180,E1 -20719.188,E2 -20719.188} C_VEL
LIN {X 0,Y 213.844,Z 603.836,A -85,B 0,C 180,E1 -20723.228,E2 -20723.228} C_VEL
LIN {X 0,Y 213.826,Z 603.851,A -85,B 0,C 180,E1 -20727.45,E2 -20727.45} C_VEL
LIN {X 0,Y 213.777,Z 603.853,A -85,B 0,C 180,E1 -20731.736,E2 -20731.736} C_VEL
LIN {X 0,Y 214.694,Z 606.583,A -85,B 0,C 180,E1 -20732.206,E2 -20732.206} C_VEL
LIN {X 0,Y 216.819,Z 608.832,A -85,B 0,C 180,E1 -20733.022,E2 -20733.022} C_VEL
LIN {X 0,Y 217.452,Z 609.512,A -85,B 0,C 180,E1 -20733.259,E2 -20733.259} C_VEL
LIN {X 0,Y 219.536,Z 612.78,A -85,B 0,C 180,E1 -20734.073,E2 -20734.073} C_VEL
LIN {X 0,Y 221.155,Z 614.68,A -85,B 0,C 180,E1 -20734.654,E2 -20734.654} C_VEL
LIN {X 0,Y 225.315,Z 620.609,A -85,B 0,C 180,E1 -20736.129,E2 -20736.129} C_VEL
LIN {X 0,Y 231.858,Z 630.246,A -85,B 0,C 180,E1 -20738.276,E2 -20738.276} C_VEL
LIN {X 0,Y 239.787,Z 643.584,A -85,B 0,C 180,E1 -20740.687,E2 -20740.687} C_VEL
LIN {X 0,Y 245.124,Z 653.62,A -85,B 0,C 180,E1 -20742.212,E2 -20742.212} C_VEL
LIN {X 0,Y 243.118,Z 695.557,A -85,B 0,C 180,E1 -20743.424,E2 -20743.424} C_VEL
LIN {X 0,Y 242.152,Z 708.911,A -85,B 0,C 180,E1 -20744.081,E2 -20744.081} C_VEL
LIN {X 0,Y 240.592,Z 721.128,A -85,B 0,C 180,E1 -20744.966,E2 -20744.966} C_VEL
LIN {X 0,Y 238.449,Z 733.096,A -85,B 0,C 180,E1 -20746.162,E2 -20746.162} C_VEL
LIN {X 0,Y 235.923,Z 744.222,A -85,B 0,C 180,E1 -20747.627,E2 -20747.627} C_VEL
LIN {X 0,Y 233.109,Z 754.352,A -85,B 0,C 180,E1 -20749.311,E2 -20749.311} C_VEL
LIN {X 0,Y 230.108,Z 763.592,A -85,B 0,C 180,E1 -20751.237,E2 -20751.237} C_VEL
LIN {X 0,Y 226.69,Z 772.876,A -85,B 0,C 180,E1 -20753.714,E2 -20753.714} C_VEL
LIN {X 0,Y 223.809,Z 780.005,A -85,B 0,C 180,E1 -20756.126,E2 -20756.126} C_VEL
LIN {X 0,Y 221.36,Z 785.432,A -85,B 0,C 180,E1 -20758.409,E2 -20758.409} C_VEL
LIN {X 0,Y 218.84,Z 790.668,A -85,B 0,C 180,E1 -20761.203,E2 -20761.203} C_VEL
LIN {X 0,Y 216.775,Z 794.657,A -85,B 0,C 180,E1 -20764.045,E2 -20764.045} C_VEL
LIN {X 0,Y 215.14,Z 797.536,A -85,B 0,C 180,E1 -20766.921,E2 -20766.921} C_VEL
LIN {X 0,Y 214.202,Z 798.875,A -85,B 0,C 180,E1 -20768.844,E2 -20768.844} C_VEL
LIN {X 0,Y 212.975,Z 800.317,A -85,B 0,C 180,E1 -20772.723,E2 -20772.723} C_VEL
LIN {X 0,Y 212.591,Z 800.4,A -85,B 0,C 180,E1 -20774.665,E2 -20774.665} C_VEL
LIN {X 0,Y 212.206,Z 799.359,A -85,B 0,C 180,E1 -20778.539,E2 -20778.539} C_VEL
LIN {X 0,Y 212.274,Z 798.233,A -85,B 0,C 180,E1 -20780.472,E2 -20780.472} C_VEL
LIN {X 0,Y 212.499,Z 796.247,A -85,B 0,C 180,E1 -20782.836,E2 -20782.836} C_VEL
LIN {X 0,Y 213.184,Z 792.255,A -85,B 0,C 180,E1 -20786.22,E2 -20786.22} C_VEL
LIN {X 0,Y 213.975,Z 787.685,A -85,B 0,C 180,E1 -20789.059,E2 -20789.059} C_VEL
LIN {X 0,Y 215.402,Z 780.779,A -85,B 0,C 180,E1 -20792.337,E2 -20792.337} C_VEL
LIN {X 0,Y 216.992,Z 773.298,A -85,B 0,C 180,E1 -20795.11,E2 -20795.11} C_VEL
LIN {X 0,Y 219.003,Z 763.876,A -85,B 0,C 180,E1 -20797.839,E2 -20797.839} C_VEL
LIN {X 0,Y 220.897,Z 754.194,A -85,B 0,C 180,E1 -20800.078,E2 -20800.078} C_VEL
LIN {X 0,Y 222.752,Z 743.563,A -85,B 0,C 180,E1 -20802.02,E2 -20802.02} C_VEL
LIN {X 0,Y 224.567,Z 731.795,A -85,B 0,C 180,E1 -20803.695,E2 -20803.695} C_VEL
LIN {X 0,Y 226.074,Z 719.55,A -85,B 0,C 180,E1 -20805.01,E2 -20805.01} C_VEL
LIN {X 0,Y 227.154,Z 705.897,A -85,B 0,C 180,E1 -20806.06,E2 -20806.06} C_VEL
LIN {X 0,Y 227.762,Z 692.991,A -85,B 0,C 180,E1 -20806.685,E2 -20806.685} C_VEL
LIN {X 0,Y 228.056,Z 681.016,A -85,B 0,C 180,E1 -20807.068,E2 -20807.068} C_VEL
LIN {X 0,Y 227.893,Z 679.324,A -85,B 0,C 180,E1 -20807.145,E2 -20807.145} C_VEL
LIN {X 0,Y 226.964,Z 700.379,A -85,B 0,C 180,E1 -20808.013,E2 -20808.013} C_VEL
LIN {X 0,Y 226.181,Z 712.2,A -85,B 0,C 180,E1 -20808.806,E2 -20808.806} C_VEL
LIN {X 0,Y 224.767,Z 725.318,A -85,B 0,C 180,E1 -20810.041,E2 -20810.041} C_VEL
LIN {X 0,Y 223.23,Z 737.151,A -85,B 0,C 180,E1 -20811.529,E2 -20811.529} C_VEL
LIN {X 0,Y 221.475,Z 748.421,A -85,B 0,C 180,E1 -20813.344,E2 -20813.344} C_VEL
LIN {X 0,Y 219.483,Z 759.485,A -85,B 0,C 180,E1 -20815.606,E2 -20815.606} C_VEL
LIN {X 0,Y 217.795,Z 768.467,A -85,B 0,C 180,E1 -20817.897,E2 -20817.897} C_VEL
LIN {X 0,Y 216.231,Z 775.995,A -85,B 0,C 180,E1 -20820.25,E2 -20820.25} C_VEL
LIN {X 0,Y 214.695,Z 783.82,A -85,B 0,C 180,E1 -20823.335,E2 -20823.335} C_VEL
LIN {X 0,Y 213.604,Z 789.737,A -85,B 0,C 180,E1 -20826.315,E2 -20826.315} C_VEL
LIN {X 0,Y 212.721,Z 794.767,A -85,B 0,C 180,E1 -20829.665,E2 -20829.665} C_VEL
LIN {X 0,Y 212.198,Z 798.469,A -85,B 0,C 180,E1 -20833.227,E2 -20833.227} C_VEL
LIN {X 0,Y 212.206,Z 800.697,A -85,B 0,C 180,E1 -20836.769,E2 -20836.769} C_VEL
LIN {X 0,Y 212.541,Z 801.421,A -85,B 0,C 180,E1 -20839.509,E2 -20839.509} C_VEL
LIN {X 0,Y 213.223,Z 801.302,A -85,B 0,C 180,E1 -20842.283,E2 -20842.283} C_VEL
LIN {X 0,Y 214.287,Z 800.305,A -85,B 0,C 180,E1 -20845.076,E2 -20845.076} C_VEL
LIN {X 0,Y 216.093,Z 797.722,A -85,B 0,C 180,E1 -20848.643,E2 -20848.643} C_VEL
LIN {X 0,Y 218.543,Z 793.425,A -85,B 0,C 180,E1 -20852.206,E2 -20852.206} C_VEL
LIN {X 0,Y 221.125,Z 788.419,A -85,B 0,C 180,E1 -20855.145,E2 -20855.145} C_VEL
LIN {X 0,Y 224.074,Z 782.252,A -85,B 0,C 180,E1 -20857.891,E2 -20857.891} C_VEL
LIN {X 0,Y 227.457,Z 774.365,A -85,B 0,C 180,E1 -20860.581,E2 -20860.581} C_VEL
LIN {X 0,Y 230.874,Z 765.485,A -85,B 0,C 180,E1 -20862.963,E2 -20862.963} C_VEL
LIN {X 0,Y 234.157,Z 755.813,A -85,B 0,C 180,E1 -20865.012,E2 -20865.012} C_VEL
LIN {X 0,Y 237.282,Z 744.912,A -85,B 0,C 180,E1 -20866.825,E2 -20866.825} C_VEL
LIN {X 0,Y 239.966,Z 733.681,A -85,B 0,C 180,E1 -20868.288,E2 -20868.288} C_VEL
LIN {X 0,Y 242.075,Z 722.495,A -85,B 0,C 180,E1 -20869.417,E2 -20869.417} C_VEL
LIN {X 0,Y 243.815,Z 709.245,A -85,B 0,C 180,E1 -20870.41,E2 -20870.41} C_VEL
LIN {X 0,Y 244.889,Z 696.571,A -85,B 0,C 180,E1 -20871.046,E2 -20871.046} C_VEL
LIN {X 0,Y 247.901,Z 654.052,A -85,B 0,C 180,E1 -20872.528,E2 -20872.528} C_VEL
LIN {X 0,Y 242.112,Z 642.987,A -85,B 0,C 180,E1 -20874.73,E2 -20874.73} C_VEL
LIN {X 0,Y 237.745,Z 635.533,A -85,B 0,C 180,E1 -20876.561,E2 -20876.561} C_VEL
LIN {X 0,Y 234.974,Z 631.536,A -85,B 0,C 180,E1 -20877.76,E2 -20877.76} C_VEL
LIN {X 0,Y 231.61,Z 627.971,A -85,B 0,C 180,E1 -20879.284,E2 -20879.284} C_VEL
LIN {X 0,Y 228.035,Z 625.51,A -85,B 0,C 180,E1 -20880.941,E2 -20880.941} C_VEL
LIN {X 0,Y 221.376,Z 621.854,A -85,B 0,C 180,E1 -20884.547,E2 -20884.547} C_VEL
LIN {X 0,Y 218.698,Z 619.501,A -85,B 0,C 180,E1 -20886.403,E2 -20886.403} C_VEL
LIN {X 0,Y 217.007,Z 616.31,A -85,B 0,C 180,E1 -20887.911,E2 -20887.911} C_VEL
LIN {X 0,Y 214.141,Z 614.209,A -85,B 0,C 180,E1 -20890.513,E2 -20890.513} C_VEL
LIN {X 0,Y 212.557,Z 611.349,A -85,B 0,C 180,E1 -20892.593,E2 -20892.593} C_VEL
LIN {X 0,Y 212.383,Z 610.727,A -85,B 0,C 180,E1 -20892.907,E2 -20892.907} C_VEL
LIN {X 0,Y 208.986,Z 609.045,A -85,B 0,C 180,E1 -20899.68,E2 -20899.68} C_VEL
LIN {X 0,Y 208.693,Z 608.92,A -85,B 0,C 180,E1 -20902.387,E2 -20902.387} C_VEL
LIN {X 0,Y 209.423,Z 611.023,A -85,B 0,C 180,E1 -20907.209,E2 -20907.209} C_VEL
LIN {X 0,Y 210.769,Z 613.457,A -85,B 0,C 180,E1 -20910.241,E2 -20910.241} C_VEL
LIN {X 0,Y 215.218,Z 619.633,A -85,B 0,C 180,E1 -20915.762,E2 -20915.762} C_VEL
LIN {X 0,Y 220.492,Z 628.028,A -85,B 0,C 180,E1 -20920.176,E2 -20920.176} C_VEL
LIN {X 0,Y 224.779,Z 635.336,A -85,B 0,C 180,E1 -20923,E2 -20923} C_VEL
LIN {X 0,Y 228.291,Z 641.602,A -85,B 0,C 180,E1 -20925.006,E2 -20925.006} C_VEL
LIN {X 0,Y 231.393,Z 647.879,A -85,B 0,C 180,E1 -20926.667,E2 -20926.667} C_VEL
LIN {X 0,Y 234.964,Z 655.451,A -85,B 0,C 180,E1 -20928.398,E2 -20928.398} C_VEL
LIN {X 0,Y 238.837,Z 665.273,A -85,B 0,C 180,E1 -20930.222,E2 -20930.222} C_VEL
LIN {X 0,Y 239.974,Z 677.653,A -85,B 0,C 180,E1 -20931.253,E2 -20931.253} C_VEL
LIN {X 0,Y 240.723,Z 694.723,A -85,B 0,C 180,E1 -20932.404,E2 -20932.404} C_VEL
LIN {X 0,Y 237.857,Z 730.273,A -85,B 0,C 180,E1 -20933.663,E2 -20933.663} C_VEL
LIN {X 0,Y 235.826,Z 744.529,A -85,B 0,C 180,E1 -20934.471,E2 -20934.471} C_VEL
LIN {X 0,Y 233.396,Z 756.064,A -85,B 0,C 180,E1 -20935.365,E2 -20935.365} C_VEL
LIN {X 0,Y 230.134,Z 768.39,A -85,B 0,C 180,E1 -20936.655,E2 -20936.655} C_VEL
LIN {X 0,Y 226.706,Z 779.556,A -85,B 0,C 180,E1 -20938.197,E2 -20938.197} C_VEL
LIN {X 0,Y 223.05,Z 789.798,A -85,B 0,C 180,E1 -20939.988,E2 -20939.988} C_VEL
LIN {X 0,Y 219.095,Z 799.94,A -85,B 0,C 180,E1 -20942.283,E2 -20942.283} C_VEL
LIN {X 0,Y 215.284,Z 808.979,A -85,B 0,C 180,E1 -20944.889,E2 -20944.889} C_VEL
LIN {X 0,Y 212.124,Z 816.376,A -85,B 0,C 180,E1 -20947.604,E2 -20947.604} C_VEL
LIN {X 0,Y 209.659,Z 822.369,A -85,B 0,C 180,E1 -20950.415,E2 -20950.415} C_VEL
LIN {X 0,Y 207.523,Z 827.18,A -85,B 0,C 180,E1 -20953.27,E2 -20953.27} C_VEL
LIN {X 0,Y 205.956,Z 830.934,A -85,B 0,C 180,E1 -20956.181,E2 -20956.181} C_VEL
LIN {X 0,Y 204.96,Z 834.42,A -85,B 0,C 180,E1 -20960.128,E2 -20960.128} C_VEL
LIN {X 0,Y 204.858,Z 836.334,A -85,B 0,C 180,E1 -20964.093,E2 -20964.093} C_VEL
LIN {X 0,Y 205.23,Z 836.565,A -85,B 0,C 180,E1 -20968.038,E2 -20968.038} C_VEL
LIN {X 0,Y 205.487,Z 836.069,A -85,B 0,C 180,E1 -20970,E2 -20970} C_VEL
LIN {X 0,Y 205.295,Z 835.536,A -85,B 0,C 180,E1 -20971.962,E2 -20971.962} C_VEL
LIN {X 0,Y 204.994,Z 835.648,A -85,B 0,C 180,E1 -20973.932,E2 -20973.932} C_VEL
LIN {X 0,Y 204.858,Z 835.323,A -85,B 0,C 180,E1 -20975.907,E2 -20975.907} C_VEL
LIN {X 0,Y 204.953,Z 833.497,A -85,B 0,C 180,E1 -20979.872,E2 -20979.872} C_VEL
LIN {X 0,Y 205.362,Z 831.992,A -85,B 0,C 180,E1 -20981.849,E2 -20981.849} C_VEL
LIN {X 0,Y 206.453,Z 828.922,A -85,B 0,C 180,E1 -20984.792,E2 -20984.792} C_VEL
LIN {X 0,Y 208.101,Z 824.827,A -85,B 0,C 180,E1 -20987.694,E2 -20987.694} C_VEL
LIN {X 0,Y 210.406,Z 819.194,A -85,B 0,C 180,E1 -20990.729,E2 -20990.729} C_VEL
LIN {X 0,Y 213.51,Z 811.801,A -85,B 0,C 180,E1 -20993.779,E2 -20993.779} C_VEL
LIN {X 0,Y 217.015,Z 803.446,A -85,B 0,C 180,E1 -20996.441,E2 -20996.441} C_VEL
LIN {X 0,Y 220.38,Z 794.859,A -85,B 0,C 180,E1 -20998.577,E2 -20998.577} C_VEL
LIN {X 0,Y 224.065,Z 784.315,A -85,B 0,C 180,E1 -21000.643,E2 -21000.643} C_VEL
LIN {X 0,Y 227.317,Z 773.872,A -85,B 0,C 180,E1 -21002.229,E2 -21002.229} C_VEL
LIN {X 0,Y 230.371,Z 762.278,A -85,B 0,C 180,E1 -21003.568,E2 -21003.568} C_VEL
LIN {X 0,Y 233.116,Z 749.045,A -85,B 0,C 180,E1 -21004.683,E2 -21004.683} C_VEL
LIN {X 0,Y 234.942,Z 736.083,A -85,B 0,C 180,E1 -21005.438,E2 -21005.438} C_VEL
LIN {X 0,Y 236.065,Z 721.759,A -85,B 0,C 180,E1 -21005.941,E2 -21005.941} C_VEL
LIN {X 0,Y 237.576,Z 689.907,A -85,B 0,C 180,E1 -21006.889,E2 -21006.889} C_VEL
LIN {X 0,Y 235.985,Z 667.924,A -85,B 0,C 180,E1 -21008.122,E2 -21008.122} C_VEL
LIN {X 0,Y 234.931,Z 657.306,A -85,B 0,C 180,E1 -21008.799,E2 -21008.799} C_VEL
LIN {X 0,Y 228.071,Z 638.942,A -85,B 0,C 180,E1 -21011.257,E2 -21011.257} C_VEL
LIN {X 0,Y 225.563,Z 633.01,A -85,B 0,C 180,E1 -21012.186,E2 -21012.186} C_VEL
LIN {X 0,Y 218.226,Z 621.84,A -85,B 0,C 180,E1 -21014.833,E2 -21014.833} C_VEL
LIN {X 0,Y 212.354,Z 613.576,A -85,B 0,C 180,E1 -21017.173,E2 -21017.173} C_VEL
LIN {X 0,Y 210.13,Z 610.349,A -85,B 0,C 180,E1 -21018.132,E2 -21018.132} C_VEL
LIN {X 0,Y 209.161,Z 609.23,A -85,B 0,C 180,E1 -21018.547,E2 -21018.547} C_VEL
LIN {X 0,Y 207.582,Z 607.315,A -85,B 0,C 180,E1 -21019.365,E2 -21019.365} C_VEL
LIN {X 0,Y 206.726,Z 604.717,A -85,B 0,C 180,E1 -21020.168,E2 -21020.168} C_VEL
LIN {X 0,Y 206.729,Z 604.714,A -85,B 0,C 180,E1 -21024.694,E2 -21024.694} C_VEL
LIN {X 0,Y 206.704,Z 604.724,A -85,B 0,C 180,E1 -21029.336,E2 -21029.336} C_VEL
LIN {X 0,Y 206.73,Z 604.733,A -85,B 0,C 180,E1 -21033.772,E2 -21033.772} C_VEL
LIN {X 0,Y 206.753,Z 604.705,A -85,B 0,C 180,E1 -21038.043,E2 -21038.043} C_VEL
LIN {X 0,Y 206.872,Z 604.701,A -85,B 0,C 180,E1 -21042.196,E2 -21042.196} C_VEL
LIN {X 0,Y 206.888,Z 604.703,A -85,B 0,C 180,E1 -21046.244,E2 -21046.244} C_VEL
LIN {X 0,Y 207.095,Z 604.66,A -85,B 0,C 180,E1 -21050.231,E2 -21050.231} C_VEL
LIN {X 0,Y 207.059,Z 604.691,A -85,B 0,C 180,E1 -21054.156,E2 -21054.156} C_VEL
LIN {X 0,Y 207.378,Z 604.622,A -85,B 0,C 180,E1 -21058.058,E2 -21058.058} C_VEL
LIN {X 0,Y 207.51,Z 604.615,A -85,B 0,C 180,E1 -21060,E2 -21060} C_VEL
LIN {X 0,Y 207.379,Z 604.653,A -85,B 0,C 180,E1 -21061.942,E2 -21061.942} C_VEL
LIN {X 0,Y 207.162,Z 604.667,A -85,B 0,C 180,E1 -21067.799,E2 -21067.799} C_VEL
LIN {X 0,Y 206.938,Z 604.683,A -85,B 0,C 180,E1 -21071.758,E2 -21071.758} C_VEL
LIN {X 0,Y 206.863,Z 604.718,A -85,B 0,C 180,E1 -21075.771,E2 -21075.771} C_VEL
LIN {X 0,Y 206.779,Z 604.707,A -85,B 0,C 180,E1 -21079.87,E2 -21079.87} C_VEL
LIN {X 0,Y 206.76,Z 604.711,A -85,B 0,C 180,E1 -21084.073,E2 -21084.073} C_VEL
LIN {X 0,Y 206.721,Z 604.719,A -85,B 0,C 180,E1 -21089.186,E2 -21089.186} C_VEL
LIN {X 0,Y 207.754,Z 607.616,A -85,B 0,C 180,E1 -21089.792,E2 -21089.792} C_VEL
LIN {X 0,Y 209.952,Z 609.836,A -85,B 0,C 180,E1 -21090.732,E2 -21090.732} C_VEL
LIN {X 0,Y 210.569,Z 610.445,A -85,B 0,C 180,E1 -21090.988,E2 -21090.988} C_VEL
LIN {X 0,Y 212.596,Z 613.677,A -85,B 0,C 180,E1 -21091.874,E2 -21091.874} C_VEL
LIN {X 0,Y 214.307,Z 615.516,A -85,B 0,C 180,E1 -21092.55,E2 -21092.55} C_VEL
LIN {X 0,Y 216.946,Z 619.184,A -85,B 0,C 180,E1 -21093.592,E2 -21093.592} C_VEL
LIN {X 0,Y 223.18,Z 628.007,A -85,B 0,C 180,E1 -21095.879,E2 -21095.879} C_VEL
LIN {X 0,Y 230.088,Z 638.856,A -85,B 0,C 180,E1 -21098.209,E2 -21098.209} C_VEL
LIN {X 0,Y 236.872,Z 650.818,A -85,B 0,C 180,E1 -21100.329,E2 -21100.329} C_VEL
LIN {X 0,Y 239.706,Z 656.259,A -85,B 0,C 180,E1 -21101.177,E2 -21101.177} C_VEL
LIN {X 0,Y 237.698,Z 696.016,A -85,B 0,C 180,E1 -21102.34,E2 -21102.34} C_VEL
LIN {X 0,Y 236.655,Z 709.682,A -85,B 0,C 180,E1 -21103.024,E2 -21103.024} C_VEL
LIN {X 0,Y 234.948,Z 722.426,A -85,B 0,C 180,E1 -21103.974,E2 -21103.974} C_VEL
LIN {X 0,Y 232.822,Z 733.663,A -85,B 0,C 180,E1 -21105.123,E2 -21105.123} C_VEL
LIN {X 0,Y 230.181,Z 744.794,A -85,B 0,C 180,E1 -21106.61,E2 -21106.61} C_VEL
LIN {X 0,Y 227.099,Z 755.433,A -85,B 0,C 180,E1 -21108.418,E2 -21108.418} C_VEL
LIN {X 0,Y 223.772,Z 765.074,A -85,B 0,C 180,E1 -21110.508,E2 -21110.508} C_VEL
LIN {X 0,Y 220.122,Z 774.473,A -85,B 0,C 180,E1 -21113.124,E2 -21113.124} C_VEL
LIN {X 0,Y 216.689,Z 782.341,A -85,B 0,C 180,E1 -21115.981,E2 -21115.981} C_VEL
LIN {X 0,Y 213.84,Z 788.17,A -85,B 0,C 180,E1 -21118.706,E2 -21118.706} C_VEL
LIN {X 0,Y 210.924,Z 793.742,A -85,B 0,C 180,E1 -21122.195,E2 -21122.195} C_VEL
LIN {X 0,Y 208.88,Z 797.196,A -85,B 0,C 180,E1 -21125.292,E2 -21125.292} C_VEL
LIN {X 0,Y 207.418,Z 799.349,A -85,B 0,C 180,E1 -21128.117,E2 -21128.117} C_VEL
LIN {X 0,Y 206.637,Z 800.309,A -85,B 0,C 180,E1 -21130.117,E2 -21130.117} C_VEL
LIN {X 0,Y 205.86,Z 800.977,A -85,B 0,C 180,E1 -21132.924,E2 -21132.924} C_VEL
LIN {X 0,Y 205.281,Z 800.749,A -85,B 0,C 180,E1 -21136.134,E2 -21136.134} C_VEL
LIN {X 0,Y 205.179,Z 799.007,A -85,B 0,C 180,E1 -21140.139,E2 -21140.139} C_VEL
LIN {X 0,Y 205.416,Z 796.856,A -85,B 0,C 180,E1 -21142.836,E2 -21142.836} C_VEL
LIN {X 0,Y 206.077,Z 793.192,A -85,B 0,C 180,E1 -21146.089,E2 -21146.089} C_VEL
LIN {X 0,Y 206.871,Z 788.73,A -85,B 0,C 180,E1 -21149.027,E2 -21149.027} C_VEL
LIN {X 0,Y 208.322,Z 781.936,A -85,B 0,C 180,E1 -21152.417,E2 -21152.417} C_VEL
LIN {X 0,Y 209.921,Z 774.59,A -85,B 0,C 180,E1 -21155.282,E2 -21155.282} C_VEL
LIN {X 0,Y 211.632,Z 767.067,A -85,B 0,C 180,E1 -21157.633,E2 -21157.633} C_VEL
LIN {X 0,Y 213.732,Z 756.882,A -85,B 0,C 180,E1 -21160.18,E2 -21160.18} C_VEL
LIN {X 0,Y 215.722,Z 746.072,A -85,B 0,C 180,E1 -21162.321,E2 -21162.321} C_VEL
LIN {X 0,Y 217.62,Z 734.699,A -85,B 0,C 180,E1 -21164.056,E2 -21164.056} C_VEL
LIN {X 0,Y 219.358,Z 721.666,A -85,B 0,C 180,E1 -21165.564,E2 -21165.564} C_VEL
LIN {X 0,Y 220.502,Z 709.102,A -85,B 0,C 180,E1 -21166.61,E2 -21166.61} C_VEL
LIN {X 0,Y 220.848,Z 701.221,A -85,B 0,C 180,E1 -21167.103,E2 -21167.103} C_VEL
LIN {X 0,Y 220.443,Z 699.12,A -85,B 0,C 180,E1 -21167.285,E2 -21167.285} C_VEL
LIN {X 0,Y 219.63,Z 711.497,A -85,B 0,C 180,E1 -21168.102,E2 -21168.102} C_VEL
LIN {X 0,Y 218.282,Z 723.972,A -85,B 0,C 180,E1 -21169.25,E2 -21169.25} C_VEL
LIN {X 0,Y 216.78,Z 735.556,A -85,B 0,C 180,E1 -21170.691,E2 -21170.691} C_VEL
LIN {X 0,Y 214.903,Z 747.514,A -85,B 0,C 180,E1 -21172.597,E2 -21172.597} C_VEL
LIN {X 0,Y 213.039,Z 757.55,A -85,B 0,C 180,E1 -21174.612,E2 -21174.612} C_VEL
LIN {X 0,Y 211.181,Z 767.102,A -85,B 0,C 180,E1 -21177.012,E2 -21177.012} C_VEL
LIN {X 0,Y 209.368,Z 775.876,A -85,B 0,C 180,E1 -21179.749,E2 -21179.749} C_VEL
LIN {X 0,Y 207.813,Z 783.504,A -85,B 0,C 180,E1 -21182.758,E2 -21182.758} C_VEL
LIN {X 0,Y 206.614,Z 789.767,A -85,B 0,C 180,E1 -21185.925,E2 -21185.925} C_VEL
LIN {X 0,Y 205.721,Z 794.912,A -85,B 0,C 180,E1 -21189.336,E2 -21189.336} C_VEL
LIN {X 0,Y 205.353,Z 797.032,A -85,B 0,C 180,E1 -21191.155,E2 -21191.155} C_VEL
LIN {X 0,Y 205.075,Z 799.566,A -85,B 0,C 180,E1 -21193.972,E2 -21193.972} C_VEL
LIN {X 0,Y 205.122,Z 801.188,A -85,B 0,C 180,E1 -21196.744,E2 -21196.744} C_VEL
LIN {X 0,Y 205.448,Z 802.001,A -85,B 0,C 180,E1 -21199.462,E2 -21199.462} C_VEL
LIN {X 0,Y 206.1,Z 802.069,A -85,B 0,C 180,E1 -21202.135,E2 -21202.135} C_VEL
LIN {X 0,Y 207.064,Z 801.404,A -85,B 0,C 180,E1 -21204.76,E2 -21204.76} C_VEL
LIN {X 0,Y 208.337,Z 799.896,A -85,B 0,C 180,E1 -21207.493,E2 -21207.493} C_VEL
LIN {X 0,Y 210.111,Z 797.33,A -85,B 0,C 180,E1 -21210.418,E2 -21210.418} C_VEL
LIN {X 0,Y 212.323,Z 793.654,A -85,B 0,C 180,E1 -21213.341,E2 -21213.341} C_VEL
LIN {X 0,Y 215.019,Z 788.742,A -85,B 0,C 180,E1 -21216.23,E2 -21216.23} C_VEL
LIN {X 0,Y 218.48,Z 781.854,A -85,B 0,C 180,E1 -21219.277,E2 -21219.277} C_VEL
LIN {X 0,Y 222.21,Z 773.586,A -85,B 0,C 180,E1 -21222.068,E2 -21222.068} C_VEL
LIN {X 0,Y 225.532,Z 765.413,A -85,B 0,C 180,E1 -21224.226,E2 -21224.226} C_VEL
LIN {X 0,Y 229.101,Z 755.075,A -85,B 0,C 180,E1 -21226.39,E2 -21226.39} C_VEL
LIN {X 0,Y 232.437,Z 743.832,A -85,B 0,C 180,E1 -21228.223,E2 -21228.223} C_VEL
LIN {X 0,Y 235.215,Z 732.37,A -85,B 0,C 180,E1 -21229.672,E2 -21229.672} C_VEL
LIN {X 0,Y 237.636,Z 719.372,A -85,B 0,C 180,E1 -21230.918,E2 -21230.918} C_VEL
LIN {X 0,Y 239.246,Z 706.482,A -85,B 0,C 180,E1 -21231.817,E2 -21231.817} C_VEL
LIN {X 0,Y 240.421,Z 692.058,A -85,B 0,C 180,E1 -21232.439,E2 -21232.439} C_VEL
LIN {X 0,Y 243.074,Z 656.946,A -85,B 0,C 180,E1 -21233.665,E2 -21233.665} C_VEL
LIN {X 0,Y 237.335,Z 645.979,A -85,B 0,C 180,E1 -21236.036,E2 -21236.036} C_VEL
LIN {X 0,Y 233.412,Z 639.286,A -85,B 0,C 180,E1 -21237.798,E2 -21237.798} C_VEL
LIN {X 0,Y 227.154,Z 629.818,A -85,B 0,C 180,E1 -21240.982,E2 -21240.982} C_VEL
LIN {X 0,Y 224.563,Z 626.069,A -85,B 0,C 180,E1 -21242.512,E2 -21242.512} C_VEL
LIN {X 0,Y 221.752,Z 622.455,A -85,B 0,C 180,E1 -21244.274,E2 -21244.274} C_VEL
LIN {X 0,Y 221.376,Z 621.854,A -85,B 0,C 180,E1 -21244.547,E2 -21244.547} C_VEL
LIN {X 0,Y 219.328,Z 621.402,A -85,B 0,C 180,E1 -21245.817,E2 -21245.817} C_VEL
LIN {X 0,Y 214.874,Z 622.498,A -85,B 0,C 180,E1 -21248.77,E2 -21248.77} C_VEL
LIN {X 0,Y 213.694,Z 622.045,A -85,B 0,C 180,E1 -21249.782,E2 -21249.782} C_VEL
LIN {X 0,Y 211.65,Z 619.519,A -85,B 0,C 180,E1 -21252.13,E2 -21252.13} C_VEL
LIN {X 0,Y 210.774,Z 617.62,A -85,B 0,C 180,E1 -21253.498,E2 -21253.498} C_VEL
LIN {X 0,Y 207.861,Z 616.048,A -85,B 0,C 180,E1 -21259.762,E2 -21259.762} C_VEL
LIN {X 0,Y 207.579,Z 615.905,A -85,B 0,C 180,E1 -21262.189,E2 -21262.189} C_VEL
LIN {X 0,Y 208.161,Z 617.875,A -85,B 0,C 180,E1 -21266.803,E2 -21266.803} C_VEL
LIN {X 0,Y 209.355,Z 620.186,A -85,B 0,C 180,E1 -21269.759,E2 -21269.759} C_VEL
LIN {X 0,Y 213.414,Z 626.166,A -85,B 0,C 180,E1 -21275.168,E2 -21275.168} C_VEL
LIN {X 0,Y 218.227,Z 634.232,A -85,B 0,C 180,E1 -21279.473,E2 -21279.473} C_VEL
LIN {X 0,Y 222.312,Z 641.545,A -85,B 0,C 180,E1 -21282.339,E2 -21282.339} C_VEL
LIN {X 0,Y 225.511,Z 647.644,A -85,B 0,C 180,E1 -21284.309,E2 -21284.309} C_VEL
LIN {X 0,Y 228.598,Z 654.174,A -85,B 0,C 180,E1 -21286.047,E2 -21286.047} C_VEL
LIN {X 0,Y 231.693,Z 661.196,A -85,B 0,C 180,E1 -21287.667,E2 -21287.667} C_VEL
LIN {X 0,Y 234.667,Z 669.255,A -85,B 0,C 180,E1 -21289.17,E2 -21289.17} C_VEL
LIN {X 0,Y 235.727,Z 686.353,A -85,B 0,C 180,E1 -21290.543,E2 -21290.543} C_VEL
LIN {X 0,Y 235.918,Z 696.485,A -85,B 0,C 180,E1 -21291.181,E2 -21291.181} C_VEL
LIN {X 0,Y 233.037,Z 730.22,A -85,B 0,C 180,E1 -21292.398,E2 -21292.398} C_VEL
LIN {X 0,Y 230.956,Z 744.041,A -85,B 0,C 180,E1 -21293.196,E2 -21293.196} C_VEL
LIN {X 0,Y 228.155,Z 756.404,A -85,B 0,C 180,E1 -21294.179,E2 -21294.179} C_VEL
LIN {X 0,Y 224.775,Z 768.458,A -85,B 0,C 180,E1 -21295.48,E2 -21295.48} C_VEL
LIN {X 0,Y 221.17,Z 779.434,A -85,B 0,C 180,E1 -21297.033,E2 -21297.033} C_VEL
LIN {X 0,Y 217.366,Z 789.537,A -85,B 0,C 180,E1 -21298.848,E2 -21298.848} C_VEL
LIN {X 0,Y 213.604,Z 798.779,A -85,B 0,C 180,E1 -21300.968,E2 -21300.968} C_VEL
LIN {X 0,Y 209.491,Z 807.902,A -85,B 0,C 180,E1 -21303.609,E2 -21303.609} C_VEL
LIN {X 0,Y 206.059,Z 815.338,A -85,B 0,C 180,E1 -21306.375,E2 -21306.375} C_VEL
LIN {X 0,Y 202.955,Z 822.243,A -85,B 0,C 180,E1 -21309.74,E2 -21309.74} C_VEL
LIN {X 0,Y 200.689,Z 826.937,A -85,B 0,C 180,E1 -21312.683,E2 -21312.683} C_VEL
LIN {X 0,Y 199.031,Z 830.585,A -85,B 0,C 180,E1 -21315.69,E2 -21315.69} C_VEL
LIN {X 0,Y 197.924,Z 833.955,A -85,B 0,C 180,E1 -21319.774,E2 -21319.774} C_VEL
LIN {X 0,Y 197.709,Z 835.051,A -85,B 0,C 180,E1 -21321.826,E2 -21321.826} C_VEL
LIN {X 0,Y 197.803,Z 835.784,A -85,B 0,C 180,E1 -21324.183,E2 -21324.183} C_VEL
LIN {X 0,Y 198.141,Z 835.861,A -85,B 0,C 180,E1 -21327.967,E2 -21327.967} C_VEL
LIN {X 0,Y 198.433,Z 835.322,A -85,B 0,C 180,E1 -21330,E2 -21330} C_VEL
LIN {X 0,Y 198.199,Z 834.891,A -85,B 0,C 180,E1 -21332.032,E2 -21332.032} C_VEL
LIN {X 0,Y 197.785,Z 834.84,A -85,B 0,C 180,E1 -21335.765,E2 -21335.765} C_VEL
LIN {X 0,Y 197.705,Z 834.057,A -85,B 0,C 180,E1 -21338.174,E2 -21338.174} C_VEL
LIN {X 0,Y 198.385,Z 831.516,A -85,B 0,C 180,E1 -21342.272,E2 -21342.272} C_VEL
LIN {X 0,Y 199.565,Z 828.495,A -85,B 0,C 180,E1 -21345.315,E2 -21345.315} C_VEL
LIN {X 0,Y 201.322,Z 824.46,A -85,B 0,C 180,E1 -21348.311,E2 -21348.311} C_VEL
LIN {X 0,Y 203.986,Z 818.346,A -85,B 0,C 180,E1 -21351.712,E2 -21351.712} C_VEL
LIN {X 0,Y 207.011,Z 811.602,A -85,B 0,C 180,E1 -21354.574,E2 -21354.574} C_VEL
LIN {X 0,Y 210.677,Z 803.347,A -85,B 0,C 180,E1 -21357.302,E2 -21357.302} C_VEL
LIN {X 0,Y 214.168,Z 794.9,A -85,B 0,C 180,E1 -21359.486,E2 -21359.486} C_VEL
LIN {X 0,Y 217.989,Z 784.49,A -85,B 0,C 180,E1 -21361.594,E2 -21361.594} C_VEL
LIN {X 0,Y 221.372,Z 774.218,A -85,B 0,C 180,E1 -21363.205,E2 -21363.205} C_VEL
LIN {X 0,Y 224.521,Z 762.98,A -85,B 0,C 180,E1 -21364.565,E2 -21364.565} C_VEL
LIN {X 0,Y 227.35,Z 750.182,A -85,B 0,C 180,E1 -21365.694,E2 -21365.694} C_VEL
LIN {X 0,Y 229.379,Z 737.137,A -85,B 0,C 180,E1 -21366.509,E2 -21366.509} C_VEL
LIN {X 0,Y 230.509,Z 724.985,A -85,B 0,C 180,E1 -21366.987,E2 -21366.987} C_VEL
LIN {X 0,Y 232.258,Z 690.871,A -85,B 0,C 180,E1 -21368.012,E2 -21368.012} C_VEL
LIN {X 0,Y 230.696,Z 667.856,A -85,B 0,C 180,E1 -21369.344,E2 -21369.344} C_VEL
LIN {X 0,Y 229.895,Z 660.064,A -85,B 0,C 180,E1 -21369.872,E2 -21369.872} C_VEL
LIN {X 0,Y 223.86,Z 643.466,A -85,B 0,C 180,E1 -21372.166,E2 -21372.166} C_VEL
LIN {X 0,Y 221.438,Z 637.592,A -85,B 0,C 180,E1 -21373.116,E2 -21373.116} C_VEL
LIN {X 0,Y 214.661,Z 627.069,A -85,B 0,C 180,E1 -21375.689,E2 -21375.689} C_VEL
LIN {X 0,Y 209.037,Z 619.063,A -85,B 0,C 180,E1 -21378.036,E2 -21378.036} C_VEL
LIN {X 0,Y 206.197,Z 615.107,A -85,B 0,C 180,E1 -21379.318,E2 -21379.318} C_VEL
LIN {X 0,Y 203.586,Z 611.633,A -85,B 0,C 180,E1 -21380.559,E2 -21380.559} C_VEL
LIN {X 0,Y 202.928,Z 610.712,A -85,B 0,C 180,E1 -21380.887,E2 -21380.887} C_VEL
LIN {X 0,Y 200.716,Z 608.466,A -85,B 0,C 180,E1 -21381.972,E2 -21381.972} C_VEL
LIN {X 0,Y 199.659,Z 605.615,A -85,B 0,C 180,E1 -21382.929,E2 -21382.929} C_VEL
LIN {X 0,Y 199.693,Z 605.611,A -85,B 0,C 180,E1 -21388.136,E2 -21388.136} C_VEL
LIN {X 0,Y 199.683,Z 605.598,A -85,B 0,C 180,E1 -21392.771,E2 -21392.771} C_VEL
LIN {X 0,Y 199.734,Z 605.577,A -85,B 0,C 180,E1 -21397.229,E2 -21397.229} C_VEL
LIN {X 0,Y 199.834,Z 605.584,A -85,B 0,C 180,E1 -21401.721,E2 -21401.721} C_VEL
LIN {X 0,Y 199.828,Z 605.574,A -85,B 0,C 180,E1 -21405.748,E2 -21405.748} C_VEL
LIN {X 0,Y 200.019,Z 605.544,A -85,B 0,C 180,E1 -21409.882,E2 -21409.882} C_VEL
LIN {X 0,Y 200.02,Z 605.566,A -85,B 0,C 180,E1 -21413.949,E2 -21413.949} C_VEL
LIN {X 0,Y 200.317,Z 605.501,A -85,B 0,C 180,E1 -21417.989,E2 -21417.989} C_VEL
LIN {X 0,Y 200.475,Z 605.49,A -85,B 0,C 180,E1 -21420,E2 -21420} C_VEL
LIN {X 0,Y 200.027,Z 605.547,A -85,B 0,C 180,E1 -21424.03,E2 -21424.03} C_VEL
LIN {X 0,Y 200.106,Z 605.549,A -85,B 0,C 180,E1 -21428.076,E2 -21428.076} C_VEL
LIN {X 0,Y 200.032,Z 605.558,A -85,B 0,C 180,E1 -21430.347,E2 -21430.347} C_VEL
LIN {X 0,Y 199.801,Z 605.595,A -85,B 0,C 180,E1 -21436.344,E2 -21436.344} C_VEL
LIN {X 0,Y 199.696,Z 605.597,A -85,B 0,C 180,E1 -21440.606,E2 -21440.606} C_VEL
LIN {X 0,Y 199.669,Z 605.593,A -85,B 0,C 180,E1 -21444.985,E2 -21444.985} C_VEL
LIN {X 0,Y 199.7,Z 605.598,A -85,B 0,C 180,E1 -21446.309,E2 -21446.309} C_VEL
LIN {X 0,Y 200.639,Z 608.384,A -85,B 0,C 180,E1 -21446.948,E2 -21446.948} C_VEL
LIN {X 0,Y 202.807,Z 610.611,A -85,B 0,C 180,E1 -21448.012,E2 -21448.012} C_VEL
LIN {X 0,Y 203.711,Z 611.286,A -85,B 0,C 180,E1 -21448.425,E2 -21448.425} C_VEL
LIN {X 0,Y 205.588,Z 614.468,A -85,B 0,C 180,E1 -21449.363,E2 -21449.363} C_VEL
LIN {X 0,Y 207.692,Z 616.691,A -85,B 0,C 180,E1 -21450.292,E2 -21450.292} C_VEL
LIN {X 0,Y 210.294,Z 620.282,A -85,B 0,C 180,E1 -21451.435,E2 -21451.435} C_VEL
LIN {X 0,Y 211.725,Z 622.274,A -85,B 0,C 180,E1 -21452.04,E2 -21452.04} C_VEL
LIN {X 0,Y 215.233,Z 627.112,A -85,B 0,C 180,E1 -21453.455,E2 -21453.455} C_VEL
LIN {X 0,Y 219.811,Z 633.742,A -85,B 0,C 180,E1 -21455.184,E2 -21455.184} C_VEL
LIN {X 0,Y 226.302,Z 644.138,A -85,B 0,C 180,E1 -21457.473,E2 -21457.473} C_VEL
LIN {X 0,Y 232.719,Z 655.648,A -85,B 0,C 180,E1 -21459.57,E2 -21459.57} C_VEL
LIN {X 0,Y 234.38,Z 658.79,A -85,B 0,C 180,E1 -21460.089,E2 -21460.089} C_VEL
LIN {X 0,Y 232.521,Z 693.806,A -85,B 0,C 180,E1 -21461.117,E2 -21461.117} C_VEL
LIN {X 0,Y 231.515,Z 707.6,A -85,B 0,C 180,E1 -21461.725,E2 -21461.725} C_VEL
LIN {X 0,Y 229.859,Z 720.544,A -85,B 0,C 180,E1 -21462.651,E2 -21462.651} C_VEL
LIN {X 0,Y 227.671,Z 732.429,A -85,B 0,C 180,E1 -21463.818,E2 -21463.818} C_VEL
LIN {X 0,Y 224.906,Z 743.972,A -85,B 0,C 180,E1 -21465.326,E2 -21465.326} C_VEL
LIN {X 0,Y 221.501,Z 755.437,A -85,B 0,C 180,E1 -21467.272,E2 -21467.272} C_VEL
LIN {X 0,Y 218.183,Z 764.78,A -85,B 0,C 180,E1 -21469.287,E2 -21469.287} C_VEL
LIN {X 0,Y 214.402,Z 774.108,A -85,B 0,C 180,E1 -21471.879,E2 -21471.879} C_VEL
LIN {X 0,Y 211.22,Z 781.2,A -85,B 0,C 180,E1 -21474.39,E2 -21474.39} C_VEL
LIN {X 0,Y 208.003,Z 787.622,A -85,B 0,C 180,E1 -21477.276,E2 -21477.276} C_VEL
LIN {X 0,Y 205.272,Z 792.616,A -85,B 0,C 180,E1 -21480.236,E2 -21480.236} C_VEL
LIN {X 0,Y 203.023,Z 796.403,A -85,B 0,C 180,E1 -21483.256,E2 -21483.256} C_VEL
LIN {X 0,Y 201.75,Z 798.32,A -85,B 0,C 180,E1 -21485.291,E2 -21485.291} C_VEL
LIN {X 0,Y 200.666,Z 799.809,A -85,B 0,C 180,E1 -21487.341,E2 -21487.341} C_VEL
LIN {X 0,Y 199.804,Z 800.823,A -85,B 0,C 180,E1 -21489.406,E2 -21489.406} C_VEL
LIN {X 0,Y 198.637,Z 801.636,A -85,B 0,C 180,E1 -21493.558,E2 -21493.558} C_VEL
LIN {X 0,Y 198.281,Z 801.421,A -85,B 0,C 180,E1 -21495.635,E2 -21495.635} C_VEL
LIN {X 0,Y 198.085,Z 799.759,A -85,B 0,C 180,E1 -21499.782,E2 -21499.782} C_VEL
LIN {X 0,Y 198.34,Z 797.475,A -85,B 0,C 180,E1 -21502.819,E2 -21502.819} C_VEL
LIN {X 0,Y 198.946,Z 794.107,A -85,B 0,C 180,E1 -21505.949,E2 -21505.949} C_VEL
LIN {X 0,Y 199.771,Z 789.734,A -85,B 0,C 180,E1 -21508.992,E2 -21508.992} C_VEL
LIN {X 0,Y 201.242,Z 783.087,A -85,B 0,C 180,E1 -21512.502,E2 -21512.502} C_VEL
LIN {X 0,Y 202.868,Z 775.855,A -85,B 0,C 180,E1 -21515.467,E2 -21515.467} C_VEL
LIN {X 0,Y 204.613,Z 768.466,A -85,B 0,C 180,E1 -21517.897,E2 -21517.897} C_VEL
LIN {X 0,Y 206.606,Z 759.533,A -85,B 0,C 180,E1 -21520.287,E2 -21520.287} C_VEL
LIN {X 0,Y 208.61,Z 749.28,A -85,B 0,C 180,E1 -21522.476,E2 -21522.476} C_VEL
LIN {X 0,Y 210.523,Z 738.547,A -85,B 0,C 180,E1 -21524.283,E2 -21524.283} C_VEL
LIN {X 0,Y 212.292,Z 726.538,A -85,B 0,C 180,E1 -21525.85,E2 -21525.85} C_VEL
LIN {X 0,Y 213.729,Z 713.474,A -85,B 0,C 180,E1 -21527.087,E2 -21527.087} C_VEL
LIN {X 0,Y 213.037,Z 711.16,A -85,B 0,C 180,E1 -21527.395,E2 -21527.395} C_VEL
LIN {X 0,Y 211.597,Z 724.493,A -85,B 0,C 180,E1 -21528.643,E2 -21528.643} C_VEL
LIN {X 0,Y 209.834,Z 737.376,A -85,B 0,C 180,E1 -21530.313,E2 -21530.313} C_VEL
LIN {X 0,Y 208.112,Z 747.932,A -85,B 0,C 180,E1 -21532.064,E2 -21532.064} C_VEL
LIN {X 0,Y 206.173,Z 758.037,A -85,B 0,C 180,E1 -21534.145,E2 -21534.145} C_VEL
LIN {X 0,Y 204.084,Z 768.468,A -85,B 0,C 180,E1 -21536.87,E2 -21536.87} C_VEL
LIN {X 0,Y 202.219,Z 777.052,A -85,B 0,C 180,E1 -21539.673,E2 -21539.673} C_VEL
LIN {X 0,Y 200.682,Z 784.586,A -85,B 0,C 180,E1 -21542.808,E2 -21542.808} C_VEL
LIN {X 0,Y 199.52,Z 790.437,A -85,B 0,C 180,E1 -21545.888,E2 -21545.888} C_VEL
LIN {X 0,Y 198.718,Z 794.921,A -85,B 0,C 180,E1 -21548.916,E2 -21548.916} C_VEL
LIN {X 0,Y 198.101,Z 798.722,A -85,B 0,C 180,E1 -21552.38,E2 -21552.38} C_VEL
LIN {X 0,Y 197.981,Z 800.864,A -85,B 0,C 180,E1 -21555.231,E2 -21555.231} C_VEL
LIN {X 0,Y 198.159,Z 802.229,A -85,B 0,C 180,E1 -21558.14,E2 -21558.14} C_VEL
LIN {X 0,Y 198.731,Z 802.784,A -85,B 0,C 180,E1 -21561.077,E2 -21561.077} C_VEL
LIN {X 0,Y 199.676,Z 802.496,A -85,B 0,C 180,E1 -21564.048,E2 -21564.048} C_VEL
LIN {X 0,Y 200.998,Z 801.299,A -85,B 0,C 180,E1 -21567.05,E2 -21567.05} C_VEL
LIN {X 0,Y 202.744,Z 799.13,A -85,B 0,C 180,E1 -21570.064,E2 -21570.064} C_VEL
LIN {X 0,Y 205.387,Z 795.229,A -85,B 0,C 180,E1 -21573.587,E2 -21573.587} C_VEL
LIN {X 0,Y 208.255,Z 790.443,A -85,B 0,C 180,E1 -21576.655,E2 -21576.655} C_VEL
LIN {X 0,Y 211.941,Z 783.737,A -85,B 0,C 180,E1 -21579.854,E2 -21579.854} C_VEL
LIN {X 0,Y 215.377,Z 776.726,A -85,B 0,C 180,E1 -21582.406,E2 -21582.406} C_VEL
LIN {X 0,Y 219.048,Z 768.266,A -85,B 0,C 180,E1 -21584.83,E2 -21584.83} C_VEL
LIN {X 0,Y 222.769,Z 758.671,A -85,B 0,C 180,E1 -21587.01,E2 -21587.01} C_VEL
LIN {X 0,Y 226.076,Z 748.746,A -85,B 0,C 180,E1 -21588.797,E2 -21588.797} C_VEL
LIN {X 0,Y 229.215,Z 737.295,A -85,B 0,C 180,E1 -21590.407,E2 -21590.407} C_VEL
LIN {X 0,Y 231.976,Z 724.608,A -85,B 0,C 180,E1 -21591.77,E2 -21591.77} C_VEL
LIN {X 0,Y 233.874,Z 712.227,A -85,B 0,C 180,E1 -21592.755,E2 -21592.755} C_VEL
LIN {X 0,Y 235.192,Z 698.796,A -85,B 0,C 180,E1 -21593.485,E2 -21593.485} C_VEL
LIN {X 0,Y 238.285,Z 659.886,A -85,B 0,C 180,E1 -21594.884,E2 -21594.884} C_VEL
LIN {X 0,Y 232.706,Z 648.985,A -85,B 0,C 180,E1 -21597.391,E2 -21597.391} C_VEL
LIN {X 0,Y 229.242,Z 643.372,A -85,B 0,C 180,E1 -21599.091,E2 -21599.091} C_VEL
LIN {X 0,Y 224.487,Z 635.746,A -85,B 0,C 180,E1 -21601.718,E2 -21601.718} C_VEL
LIN {X 0,Y 222.054,Z 632.186,A -85,B 0,C 180,E1 -21603.219,E2 -21603.219} C_VEL
LIN {X 0,Y 219.108,Z 628.264,A -85,B 0,C 180,E1 -21605.235,E2 -21605.235} C_VEL
LIN {X 0,Y 216.461,Z 625.592,A -85,B 0,C 180,E1 -21607.193,E2 -21607.193} C_VEL
LIN {X 0,Y 215.18,Z 623.03,A -85,B 0,C 180,E1 -21608.452,E2 -21608.452} C_VEL
LIN {X 0,Y 213.694,Z 622.045,A -85,B 0,C 180,E1 -21609.782,E2 -21609.782} C_VEL
LIN {X 0,Y 212.15,Z 621.292,A -85,B 0,C 180,E1 -21611.309,E2 -21611.309} C_VEL
LIN {X 0,Y 209.736,Z 621.953,A -85,B 0,C 180,E1 -21613.923,E2 -21613.923} C_VEL
LIN {X 0,Y 207.579,Z 623.321,A -85,B 0,C 180,E1 -21617.162,E2 -21617.162} C_VEL
LIN {X 0,Y 207.116,Z 623.322,A -85,B 0,C 180,E1 -21618.264,E2 -21618.264} C_VEL
LIN {X 0,Y 206.473,Z 622.888,A -85,B 0,C 180,E1 -21621.989,E2 -21621.989} C_VEL
LIN {X 0,Y 207.006,Z 624.921,A -85,B 0,C 180,E1 -21626.706,E2 -21626.706} C_VEL
LIN {X 0,Y 208.06,Z 627.126,A -85,B 0,C 180,E1 -21629.485,E2 -21629.485} C_VEL
LIN {X 0,Y 211.619,Z 632.674,A -85,B 0,C 180,E1 -21634.546,E2 -21634.546} C_VEL
LIN {X 0,Y 216.036,Z 640.483,A -85,B 0,C 180,E1 -21638.774,E2 -21638.774} C_VEL
LIN {X 0,Y 219.597,Z 647.202,A -85,B 0,C 180,E1 -21641.477,E2 -21641.477} C_VEL
LIN {X 0,Y 222.563,Z 653.149,A -85,B 0,C 180,E1 -21643.448,E2 -21643.448} C_VEL
LIN {X 0,Y 226.426,Z 661.69,A -85,B 0,C 180,E1 -21645.739,E2 -21645.739} C_VEL
LIN {X 0,Y 229.782,Z 670.501,A -85,B 0,C 180,E1 -21647.622,E2 -21647.622} C_VEL
LIN {X 0,Y 230.475,Z 672.87,A -85,B 0,C 180,E1 -21648.016,E2 -21648.016} C_VEL
LIN {X 0,Y 231.264,Z 688.709,A -85,B 0,C 180,E1 -21649.296,E2 -21649.296} C_VEL
LIN {X 0,Y 231.372,Z 697.098,A -85,B 0,C 180,E1 -21649.856,E2 -21649.856} C_VEL
LIN {X 0,Y 228.463,Z 729.344,A -85,B 0,C 180,E1 -21651.044,E2 -21651.044} C_VEL
LIN {X 0,Y 226.401,Z 742.234,A -85,B 0,C 180,E1 -21651.765,E2 -21651.765} C_VEL
LIN {X 0,Y 223.549,Z 754.914,A -85,B 0,C 180,E1 -21652.759,E2 -21652.759} C_VEL
LIN {X 0,Y 220.017,Z 767.124,A -85,B 0,C 180,E1 -21654.06,E2 -21654.06} C_VEL
LIN {X 0,Y 216.232,Z 778.219,A -85,B 0,C 180,E1 -21655.618,E2 -21655.618} C_VEL
LIN {X 0,Y 212.193,Z 788.402,A -85,B 0,C 180,E1 -21657.439,E2 -21657.439} C_VEL
LIN {X 0,Y 208.185,Z 797.671,A -85,B 0,C 180,E1 -21659.578,E2 -21659.578} C_VEL
LIN {X 0,Y 203.858,Z 806.825,A -85,B 0,C 180,E1 -21662.264,E2 -21662.264} C_VEL
